// TIA Portal project "NeuroPLC_S7_1200_DB" (V21)

(* hardware
DEVICE "PLC_1"  S7-1200 Station
   slot 0: "Rack_0"  S7-1200 Rack  Rack  V1.0
   slot 1: "PLC_1"  CPU 1211C AC/DC/Rly  6ES7 211-1BE40-0XB0  V4.7
*)

// ===== PLC "PLC_1"  CPU 1211C AC/DC/Rly =====

DATA_BLOCK "NeuroPLC_KAN_Weights"   // DB1
{ S7_Optimized_Access := 'FALSE' }
VERSION : 0.1
   VAR
      g0 : Array[0..14] of Real;   // LUT grid (15 pts)
      t1 : Array[0..6719] of Real;   // LUT table (16x28x15)
      w2 : Array[0..447] of Real;   // W(16x28)
      b3 : Array[0..15] of Real;   // bias(16)
      g4 : Array[0..14] of Real;   // LUT grid (15 pts)
      t5 : Array[0..959] of Real;   // LUT table (4x16x15)
      w6 : Array[0..63] of Real;   // W(4x16)
      b7 : Array[0..3] of Real;   // bias(4)
   END_VAR
BEGIN
   g0[0] := -3.0;
   g0[1] := -2.571429;
   g0[2] := -2.142857;
   g0[3] := -1.714286;
   g0[4] := -1.285714;
   g0[5] := -0.8571429;
   g0[6] := -0.4285714;
   g0[8] := 0.4285714;
   g0[9] := 0.8571429;
   g0[10] := 1.285714;
   g0[11] := 1.714286;
   g0[12] := 2.142857;
   g0[13] := 2.571429;
   g0[14] := 3.0;
   t1[0] := -0.1194829;
   t1[1] := -0.1267372;
   t1[2] := -0.1291282;
   t1[3] := -0.1263348;
   t1[4] := -0.1178586;
   t1[5] := -0.1031384;
   t1[6] := -0.0816128;
   t1[7] := -0.0527206;
   t1[8] := -0.0159457;
   t1[9] := 0.0269625;
   t1[10] := 0.0709812;
   t1[11] := 0.1108319;
   t1[12] := 0.141236;
   t1[13] := 0.156915;
   t1[14] := 0.1536715;
   t1[15] := -0.0048413;
   t1[16] := -0.0066063;
   t1[17] := -0.0042641;
   t1[18] := 0.0032827;
   t1[19] := 0.0154041;
   t1[20] := 0.0308592;
   t1[21] := 0.0484067;
   t1[22] := 0.0668051;
   t1[23] := 0.0848193;
   t1[24] := 0.1015272;
   t1[25] := 0.1164593;
   t1[26] := 0.1291814;
   t1[27] := 0.1392594;
   t1[28] := 0.1462591;
   t1[29] := 0.1498416;
   t1[30] := -0.08693;
   t1[31] := -0.0833493;
   t1[32] := -0.0687987;
   t1[33] := -0.0417966;
   t1[34] := -0.0053218;
   t1[35] := 0.0360709;
   t1[36] := 0.0778248;
   t1[37] := 0.1153831;
   t1[38] := 0.144237;
   t1[39] := 0.1622724;
   t1[40] := 0.1708359;
   t1[41] := 0.1715441;
   t1[42] := 0.166014;
   t1[43] := 0.1558621;
   t1[44] := 0.1426646;
   t1[45] := -0.0762567;
   t1[46] := -0.0843287;
   t1[47] := -0.0897336;
   t1[48] := -0.0919366;
   t1[49] := -0.0903113;
   t1[50] := -0.0841991;
   t1[51] := -0.0729412;
   t1[52] := -0.055879;
   t1[53] := -0.0323818;
   t1[54] := -0.0032285;
   t1[55] := 0.0287655;
   t1[56] := 0.0606256;
   t1[57] := 0.0893772;
   t1[58] := 0.1120458;
   t1[59] := 0.1260427;
   t1[60] := -0.1835549;
   t1[61] := -0.1948409;
   t1[62] := -0.1973169;
   t1[63] := -0.1890172;
   t1[64] := -0.1712564;
   t1[65] := -0.1465084;
   t1[66] := -0.1172482;
   t1[67] := -0.0859511;
   t1[68] := -0.055075;
   t1[69] := -0.0262112;
   t1[70] := 0.000301;
   t1[71] := 0.0242203;
   t1[72] := 0.0453052;
   t1[73] := 0.0633144;
   t1[74] := 0.077947;
   t1[75] := -0.0558672;
   t1[76] := -0.0577179;
   t1[77] := -0.0553535;
   t1[78] := -0.0488306;
   t1[79] := -0.0385897;
   t1[80] := -0.025207;
   t1[81] := -0.0092587;
   t1[82] := 0.008679;
   t1[83] := 0.02802;
   t1[84] := 0.0476948;
   t1[85] := 0.0659345;
   t1[86] := 0.0809157;
   t1[87] := 0.0908151;
   t1[88] := 0.0938092;
   t1[89] := 0.0884755;
   t1[90] := 0.1269326;
   t1[91] := 0.1441061;
   t1[92] := 0.1569568;
   t1[93] := 0.1633429;
   t1[94] := 0.1623842;
   t1[95] := 0.153646;
   t1[96] := 0.1366941;
   t1[97] := 0.1110945;
   t1[98] := 0.0764416;
   t1[99] := 0.0337616;
   t1[100] := -0.0138503;
   t1[101] := -0.0631375;
   t1[102] := -0.1108431;
   t1[103] := -0.1537104;
   t1[104] := -0.1886999;
   t1[105] := -0.0070284;
   t1[106] := -0.0404032;
   t1[107] := -0.064115;
   t1[108] := -0.07382;
   t1[109] := -0.0709769;
   t1[110] := -0.0590946;
   t1[111] := -0.0416847;
   t1[112] := -0.0222583;
   t1[113] := -0.0042989;
   t1[114] := 0.0101144;
   t1[115] := 0.0209318;
   t1[116] := 0.0282619;
   t1[117] := 0.0322132;
   t1[118] := 0.0328943;
   t1[119] := 0.0304549;
   t1[120] := -0.1028974;
   t1[121] := -0.1077723;
   t1[122] := -0.1036677;
   t1[123] := -0.0897878;
   t1[124] := -0.0682854;
   t1[125] := -0.0423547;
   t1[126] := -0.0151914;
   t1[127] := 0.0100092;
   t1[128] := 0.030083;
   t1[129] := 0.0434435;
   t1[130] := 0.0507842;
   t1[131] := 0.0529767;
   t1[132] := 0.0508923;
   t1[133] := 0.0454027;
   t1[134] := 0.0373401;
   t1[135] := 0.0462424;
   t1[136] := 0.0249232;
   t1[137] := 0.0137322;
   t1[138] := 0.0163544;
   t1[139] := 0.0313536;
   t1[140] := 0.0554837;
   t1[141] := 0.0854967;
   t1[142] := 0.1181446;
   t1[143] := 0.1501878;
   t1[144] := 0.1788067;
   t1[145] := 0.2017891;
   t1[146] := 0.2169701;
   t1[147] := 0.2221848;
   t1[148] := 0.2152684;
   t1[149] := 0.1947507;
   t1[150] := 0.2054697;
   t1[151] := 0.1801361;
   t1[152] := 0.1482858;
   t1[153] := 0.1121279;
   t1[154] := 0.0745698;
   t1[155] := 0.0387658;
   t1[156] := 0.0078706;
   t1[157] := -0.0149613;
   t1[158] := -0.0266352;
   t1[159] := -0.0270458;
   t1[160] := -0.0204089;
   t1[161] := -0.0112777;
   t1[162] := -0.0042051;
   t1[163] := -0.0037442;
   t1[164] := -0.0135843;
   t1[165] := 0.069604;
   t1[166] := 0.0267136;
   t1[167] := -0.0201817;
   t1[168] := -0.0687582;
   t1[169] := -0.1154626;
   t1[170] := -0.156307;
   t1[171] := -0.1873028;
   t1[172] := -0.2044615;
   t1[173] := -0.2038705;
   t1[174] := -0.1854049;
   t1[175] := -0.1544143;
   t1[176] := -0.1166757;
   t1[177] := -0.0779662;
   t1[178] := -0.0440626;
   t1[179] := -0.0199858;
   t1[180] := 0.2695681;
   t1[181] := 0.2165021;
   t1[182] := 0.1619561;
   t1[183] := 0.1091502;
   t1[184] := 0.0593546;
   t1[185] := 0.0131512;
   t1[186] := -0.0288789;
   t1[187] := -0.0661548;
   t1[188] := -0.0981051;
   t1[189] := -0.1246367;
   t1[190] := -0.146348;
   t1[191] := -0.1638913;
   t1[192] := -0.177919;
   t1[193] := -0.1890834;
   t1[194] := -0.1978753;
   t1[195] := 0.1005199;
   t1[196] := 0.1037989;
   t1[197] := 0.1110083;
   t1[198] := 0.1225618;
   t1[199] := 0.1376169;
   t1[200] := 0.1548869;
   t1[201] := 0.1730847;
   t1[202] := 0.1909233;
   t1[203] := 0.2071245;
   t1[204] := 0.2208622;
   t1[205] := 0.231963;
   t1[206] := 0.2403047;
   t1[207] := 0.2457651;
   t1[208] := 0.2482219;
   t1[209] := 0.247544;
   t1[210] := 0.0554956;
   t1[211] := 0.0007121;
   t1[212] := -0.0460094;
   t1[213] := -0.078633;
   t1[214] := -0.0985512;
   t1[215] := -0.1097806;
   t1[216] := -0.1163414;
   t1[217] := -0.1222533;
   t1[218] := -0.1314804;
   t1[219] := -0.1451906;
   t1[220] := -0.1605101;
   t1[221] := -0.1742501;
   t1[222] := -0.1832213;
   t1[223] := -0.1842349;
   t1[224] := -0.1747214;
   t1[225] := -0.0316489;
   t1[226] := -0.0383947;
   t1[227] := -0.0447371;
   t1[228] := -0.0514102;
   t1[229] := -0.0574886;
   t1[230] := -0.0614606;
   t1[231] := -0.0618138;
   t1[232] := -0.0570359;
   t1[233] := -0.045655;
   t1[234] := -0.0282333;
   t1[235] := -0.0082723;
   t1[236] := 0.010497;
   t1[237] := 0.0243434;
   t1[238] := 0.0295361;
   t1[239] := 0.0231194;
   t1[240] := -0.0541978;
   t1[241] := -0.0262211;
   t1[242] := 0.0058194;
   t1[243] := 0.0394106;
   t1[244] := 0.0729769;
   t1[245] := 0.1052741;
   t1[246] := 0.1350584;
   t1[247] := 0.161086;
   t1[248] := 0.1821203;
   t1[249] := 0.1972881;
   t1[250] := 0.2062417;
   t1[251] := 0.208674;
   t1[252] := 0.2042782;
   t1[253] := 0.1927473;
   t1[254] := 0.1740892;
   t1[255] := 0.0165106;
   t1[256] := 0.0038278;
   t1[257] := -0.0110902;
   t1[258] := -0.0267964;
   t1[259] := -0.0414656;
   t1[260] := -0.0531389;
   t1[261] := -0.059857;
   t1[262] := -0.0596609;
   t1[263] := -0.050625;
   t1[264] := -0.0325026;
   t1[265] := -0.0074732;
   t1[266] := 0.0220942;
   t1[267] := 0.0538307;
   t1[268] := 0.0853673;
   t1[269] := 0.1144174;
   t1[270] := 0.2570028;
   t1[271] := 0.2134718;
   t1[272] := 0.1650651;
   t1[273] := 0.1143154;
   t1[274] := 0.0630908;
   t1[275] := 0.0130241;
   t1[276] := -0.0342518;
   t1[277] := -0.0771044;
   t1[278] := -0.1139093;
   t1[279] := -0.1434596;
   t1[280] := -0.1651517;
   t1[281] := -0.1784292;
   t1[282] := -0.1827355;
   t1[283] := -0.1775142;
   t1[284] := -0.1625242;
   t1[285] := 0.1695031;
   t1[286] := 0.1470198;
   t1[287] := 0.1199536;
   t1[288] := 0.0881358;
   t1[289] := 0.0530191;
   t1[290] := 0.0166294;
   t1[291] := -0.0190068;
   t1[292] := -0.051863;
   t1[293] := -0.0799368;
   t1[294] := -0.1024416;
   t1[295] := -0.1203473;
   t1[296] := -0.1347608;
   t1[297] := -0.1467892;
   t1[298] := -0.1575395;
   t1[299] := -0.1678591;
   t1[300] := -0.189392;
   t1[301] := -0.1452939;
   t1[302] := -0.1035419;
   t1[303] := -0.0676707;
   t1[304] := -0.0367318;
   t1[305] := -0.0081925;
   t1[306] := 0.0204816;
   t1[307] := 0.0518252;
   t1[308] := 0.0883329;
   t1[309] := 0.1305132;
   t1[310] := 0.1760034;
   t1[311] := 0.2222168;
   t1[312] := 0.2665667;
   t1[313] := 0.3064664;
   t1[314] := 0.3394241;
   t1[315] := -0.0330082;
   t1[316] := -0.0595727;
   t1[317] := -0.0757542;
   t1[318] := -0.0766687;
   t1[319] := -0.0640394;
   t1[320] := -0.0419239;
   t1[321] := -0.0143825;
   t1[322] := 0.0145245;
   t1[323] := 0.0407725;
   t1[324] := 0.0621279;
   t1[325] := 0.0789453;
   t1[326] := 0.0917811;
   t1[327] := 0.101192;
   t1[328] := 0.1077346;
   t1[329] := 0.1118888;
   t1[330] := -0.0263191;
   t1[331] := 0.0124622;
   t1[332] := 0.0404122;
   t1[333] := 0.0524193;
   t1[334] := 0.0510294;
   t1[335] := 0.0414941;
   t1[336] := 0.0290681;
   t1[337] := 0.019006;
   t1[338] := 0.0165029;
   t1[339] := 0.0237657;
   t1[340] := 0.0386827;
   t1[341] := 0.0588053;
   t1[342] := 0.0816847;
   t1[343] := 0.1048722;
   t1[344] := 0.1260335;
   t1[345] := 0.0412466;
   t1[346] := 0.0436516;
   t1[347] := 0.0403802;
   t1[348] := 0.031226;
   t1[349] := 0.018012;
   t1[350] := 0.0032783;
   t1[351] := -0.010434;
   t1[352] := -0.0205838;
   t1[353] := -0.0246632;
   t1[354] := -0.0218213;
   t1[355] := -0.0136019;
   t1[356] := -0.0017359;
   t1[357] := 0.0120461;
   t1[358] := 0.0260132;
   t1[359] := 0.0385597;
   t1[360] := 0.1668451;
   t1[361] := 0.1318458;
   t1[362] := 0.0940298;
   t1[363] := 0.0566781;
   t1[364] := 0.0218116;
   t1[365] := -0.0089939;
   t1[366] := -0.0341632;
   t1[367] := -0.052121;
   t1[368] := -0.0613163;
   t1[369] := -0.0614061;
   t1[370] := -0.0537936;
   t1[371] := -0.0400181;
   t1[372] := -0.0216192;
   t1[373] := -0.0001363;
   t1[374] := 0.0228733;
   t1[375] := -0.2291011;
   t1[376] := -0.2048234;
   t1[377] := -0.1736495;
   t1[378] := -0.1362531;
   t1[379] := -0.0941705;
   t1[380] := -0.049243;
   t1[381] := -0.0033123;
   t1[382] := 0.0417801;
   t1[383] := 0.0841977;
   t1[384] := 0.122365;
   t1[385] := 0.1550836;
   t1[386] := 0.1811845;
   t1[387] := 0.1994988;
   t1[388] := 0.2088575;
   t1[389] := 0.2084018;
   t1[390] := 0.0971736;
   t1[391] := 0.0705846;
   t1[392] := 0.0477992;
   t1[393] := 0.0314683;
   t1[394] := 0.0213695;
   t1[395] := 0.0162659;
   t1[396] := 0.014919;
   t1[397] := 0.0160906;
   t1[398] := 0.0185539;
   t1[399] := 0.0216598;
   t1[400] := 0.0255942;
   t1[401] := 0.0306081;
   t1[402] := 0.0369525;
   t1[403] := 0.0448785;
   t1[404] := 0.0544655;
   t1[405] := 0.1530943;
   t1[406] := 0.1480777;
   t1[407] := 0.1306549;
   t1[408] := 0.0980344;
   t1[409] := 0.0543566;
   t1[410] := 0.0062115;
   t1[411] := -0.0398084;
   t1[412] := -0.0771103;
   t1[413] := -0.0991863;
   t1[414] := -0.1037752;
   t1[415] := -0.0947527;
   t1[416] := -0.0764738;
   t1[417] := -0.0532932;
   t1[418] := -0.0295659;
   t1[419] := -0.0091988;
   t1[420] := -0.1092411;
   t1[421] := -0.1059756;
   t1[422] := -0.0969084;
   t1[423] := -0.0807166;
   t1[424] := -0.0580724;
   t1[425] := -0.0303529;
   t1[426] := 0.0010639;
   t1[427] := 0.0348003;
   t1[428] := 0.0694891;
   t1[429] := 0.1043026;
   t1[430] := 0.1391932;
   t1[431] := 0.1741739;
   t1[432] := 0.2092578;
   t1[433] := 0.2444581;
   t1[434] := 0.2795447;
   t1[435] := -0.1311382;
   t1[436] := -0.1227978;
   t1[437] := -0.1088914;
   t1[438] := -0.0897558;
   t1[439] := -0.0661454;
   t1[440] := -0.0389617;
   t1[441] := -0.0091066;
   t1[442] := 0.0225182;
   t1[443] := 0.0550137;
   t1[444] := 0.0876197;
   t1[445] := 0.1197764;
   t1[446] := 0.15094;
   t1[447] := 0.1805664;
   t1[448] := 0.2081117;
   t1[449] := 0.232934;
   t1[450] := -0.2517078;
   t1[451] := -0.2631014;
   t1[452] := -0.2655013;
   t1[453] := -0.2574791;
   t1[454] := -0.2394219;
   t1[455] := -0.2123581;
   t1[456] := -0.1773168;
   t1[457] := -0.1353271;
   t1[458] := -0.0874226;
   t1[459] := -0.0348577;
   t1[460] := 0.0207941;
   t1[461] := 0.0779343;
   t1[462] := 0.1349643;
   t1[463] := 0.1902857;
   t1[464] := 0.2421744;
   t1[465] := 0.0492069;
   t1[466] := 0.0399185;
   t1[467] := 0.0213245;
   t1[468] := -0.0083821;
   t1[469] := -0.0462682;
   t1[470] := -0.0877257;
   t1[471] := -0.1281447;
   t1[472] := -0.1629154;
   t1[473] := -0.187479;
   t1[474] := -0.1998351;
   t1[475] := -0.2016807;
   t1[476] := -0.1950018;
   t1[477] := -0.181784;
   t1[478] := -0.164013;
   t1[479] := -0.1435986;
   t1[480] := 0.2468299;
   t1[481] := 0.2682943;
   t1[482] := 0.2761828;
   t1[483] := 0.2661327;
   t1[484] := 0.2398228;
   t1[485] := 0.2010666;
   t1[486] := 0.1536797;
   t1[487] := 0.1014783;
   t1[488] := 0.0482628;
   t1[489] := -0.0029272;
   t1[490] := -0.0501526;
   t1[491] := -0.0915597;
   t1[492] := -0.1252953;
   t1[493] := -0.149506;
   t1[494] := -0.1626064;
   t1[495] := -0.0399078;
   t1[496] := -0.0051029;
   t1[497] := 0.0288762;
   t1[498] := 0.0581392;
   t1[499] := 0.0810207;
   t1[500] := 0.0966417;
   t1[501] := 0.1041238;
   t1[502] := 0.1025889;
   t1[503] := 0.0911945;
   t1[504] := 0.0708923;
   t1[505] := 0.0452268;
   t1[506] := 0.0179449;
   t1[507] := -0.0072066;
   t1[508] := -0.0264807;
   t1[509] := -0.0367556;
   t1[510] := -0.227583;
   t1[511] := -0.2168898;
   t1[512] := -0.2061395;
   t1[513] := -0.197567;
   t1[514] := -0.1891667;
   t1[515] := -0.1774349;
   t1[516] := -0.1588662;
   t1[517] := -0.129955;
   t1[518] := -0.0872722;
   t1[519] := -0.0312042;
   t1[520] := 0.0323485;
   t1[521] := 0.0970544;
   t1[522] := 0.1565824;
   t1[523] := 0.2046015;
   t1[524] := 0.235604;
   t1[525] := 0.15399;
   t1[526] := 0.1505588;
   t1[527] := 0.1378421;
   t1[528] := 0.1147972;
   t1[529] := 0.084201;
   t1[530] := 0.0501803;
   t1[531] := 0.0168631;
   t1[532] := -0.0116225;
   t1[533] := -0.0311856;
   t1[534] := -0.0396094;
   t1[535] := -0.0373845;
   t1[536] := -0.0252131;
   t1[537] := -0.0037974;
   t1[538] := 0.0261603;
   t1[539] := 0.063599;
   t1[540] := -0.1692545;
   t1[541] := -0.1745036;
   t1[542] := -0.1656465;
   t1[543] := -0.1392908;
   t1[544] := -0.099259;
   t1[545] := -0.0519229;
   t1[546] := -0.0036572;
   t1[547] := 0.0391633;
   t1[548] := 0.0702438;
   t1[549] := 0.087294;
   t1[550] := 0.0938102;
   t1[551] := 0.0937407;
   t1[552] := 0.091034;
   t1[553] := 0.0896381;
   t1[554] := 0.0929436;
   t1[555] := -0.1842585;
   t1[556] := -0.1818165;
   t1[557] := -0.1727193;
   t1[558] := -0.154162;
   t1[559] := -0.126589;
   t1[560] := -0.0915928;
   t1[561] := -0.050767;
   t1[562] := -0.0057056;
   t1[563] := 0.0420004;
   t1[564] := 0.0908896;
   t1[565] := 0.1396887;
   t1[566] := 0.1871389;
   t1[567] := 0.2319812;
   t1[568] := 0.272957;
   t1[569] := 0.3087583;
   t1[570] := -0.3433722;
   t1[571] := -0.3115804;
   t1[572] := -0.2701057;
   t1[573] := -0.2195741;
   t1[574] := -0.1626008;
   t1[575] := -0.1025036;
   t1[576] := -0.0426015;
   t1[577] := 0.0137868;
   t1[578] := 0.0633724;
   t1[579] := 0.1043585;
   t1[580] := 0.1371047;
   t1[581] := 0.1621392;
   t1[582] := 0.17999;
   t1[583] := 0.1911852;
   t1[584] := 0.1962473;
   t1[585] := 0.0363517;
   t1[586] := 0.0190614;
   t1[587] := 0.0082236;
   t1[588] := 0.0071252;
   t1[589] := 0.0142321;
   t1[590] := 0.0263068;
   t1[591] := 0.0401099;
   t1[592] := 0.0524021;
   t1[593] := 0.059982;
   t1[594] := 0.0615569;
   t1[595] := 0.0585923;
   t1[596] := 0.0527691;
   t1[597] := 0.0457681;
   t1[598] := 0.0392702;
   t1[599] := 0.0347328;
   t1[600] := -0.2135215;
   t1[601] := -0.1584936;
   t1[602] := -0.0996131;
   t1[603] := -0.0401407;
   t1[604] := 0.0172358;
   t1[605] := 0.0700308;
   t1[606] := 0.1157594;
   t1[607] := 0.1519362;
   t1[608] := 0.1761245;
   t1[609] := 0.1883052;
   t1[610] := 0.1919536;
   t1[611] := 0.190818;
   t1[612] := 0.1886465;
   t1[613] := 0.1891873;
   t1[614] := 0.1954547;
   t1[615] := -0.2638247;
   t1[616] := -0.2262976;
   t1[617] := -0.181273;
   t1[618] := -0.1300747;
   t1[619] := -0.0758695;
   t1[620] := -0.0224759;
   t1[621] := 0.0262873;
   t1[622] := 0.066601;
   t1[623] := 0.0947028;
   t1[624] := 0.1096649;
   t1[625] := 0.114656;
   t1[626] := 0.1131646;
   t1[627] := 0.1086792;
   t1[628] := 0.1046883;
   t1[629] := 0.1041317;
   t1[630] := -0.0215827;
   t1[631] := -0.0225016;
   t1[632] := -0.0222959;
   t1[633] := -0.018404;
   t1[634] := -0.0125777;
   t1[635] := -0.0080928;
   t1[636] := -0.0082266;
   t1[637] := -0.0162568;
   t1[638] := -0.0353979;
   t1[639] := -0.0657176;
   t1[640] := -0.1027351;
   t1[641] := -0.1416151;
   t1[642] := -0.1775218;
   t1[643] := -0.2056196;
   t1[644] := -0.2217522;
   t1[645] := 0.0948695;
   t1[646] := 0.1189938;
   t1[647] := 0.1318502;
   t1[648] := 0.1305514;
   t1[649] := 0.1161173;
   t1[650] := 0.0909486;
   t1[651] := 0.0574476;
   t1[652] := 0.0180163;
   t1[653] := -0.0249446;
   t1[654] := -0.0691197;
   t1[655] := -0.1123164;
   t1[656] := -0.1523517;
   t1[657] := -0.1870427;
   t1[658] := -0.2142063;
   t1[659] := -0.2319627;
   t1[660] := 0.2239106;
   t1[661] := 0.2024928;
   t1[662] := 0.1690608;
   t1[663] := 0.1246878;
   t1[664] := 0.0722037;
   t1[665] := 0.0150594;
   t1[666] := -0.0432937;
   t1[667] := -0.0994042;
   t1[668] := -0.1498503;
   t1[669] := -0.1927032;
   t1[670] := -0.228191;
   t1[671] := -0.2567104;
   t1[672] := -0.278658;
   t1[673] := -0.2944305;
   t1[674] := -0.3043407;
   t1[675] := -0.210152;
   t1[676] := -0.1704469;
   t1[677] := -0.1309727;
   t1[678] := -0.0954248;
   t1[679] := -0.0645113;
   t1[680] := -0.0378848;
   t1[681] := -0.0151968;
   t1[682] := 0.0039014;
   t1[683] := 0.0197446;
   t1[684] := 0.0319798;
   t1[685] := 0.0392597;
   t1[686] := 0.0401597;
   t1[687] := 0.0332549;
   t1[688] := 0.0171205;
   t1[689] := -0.0090543;
   t1[690] := -0.2450845;
   t1[691] := -0.2073944;
   t1[692] := -0.1587359;
   t1[693] := -0.0981581;
   t1[694] := -0.0301329;
   t1[695] := 0.0389517;
   t1[696] := 0.1027057;
   t1[697] := 0.1547389;
   t1[698] := 0.1887307;
   t1[699] := 0.201844;
   t1[700] := 0.1962753;
   t1[701] := 0.1746144;
   t1[702] := 0.139451;
   t1[703] := 0.0933749;
   t1[704] := 0.0393236;
   t1[705] := -0.4248369;
   t1[706] := -0.3962753;
   t1[707] := -0.3550233;
   t1[708] := -0.3007319;
   t1[709] := -0.235328;
   t1[710] := -0.1615429;
   t1[711] := -0.0821088;
   t1[712] := 0.0002421;
   t1[713] := 0.0827594;
   t1[714] := 0.1617863;
   t1[715] := 0.2323554;
   t1[716] := 0.2893972;
   t1[717] := 0.327842;
   t1[718] := 0.3426206;
   t1[719] := 0.3299596;
   t1[720] := 0.3017888;
   t1[721] := 0.2690612;
   t1[722] := 0.2316348;
   t1[723] := 0.1906948;
   t1[724] := 0.1469425;
   t1[725] := 0.1009079;
   t1[726] := 0.0531211;
   t1[727] := 0.0041119;
   t1[728] := -0.0455605;
   t1[729] := -0.0938802;
   t1[730] := -0.136726;
   t1[731] := -0.1698123;
   t1[732] := -0.1888533;
   t1[733] := -0.1895635;
   t1[734] := -0.1688053;
   t1[735] := 0.2525824;
   t1[736] := 0.18621;
   t1[737] := 0.1176589;
   t1[738] := 0.051741;
   t1[739] := -0.0101694;
   t1[740] := -0.0679128;
   t1[741] := -0.121331;
   t1[742] := -0.1702659;
   t1[743] := -0.2145509;
   t1[744] := -0.2535933;
   t1[745] := -0.2861848;
   t1[746] := -0.3110689;
   t1[747] := -0.3269894;
   t1[748] := -0.3326899;
   t1[749] := -0.3272332;
   t1[750] := 0.1863346;
   t1[751] := 0.1608573;
   t1[752] := 0.1253638;
   t1[753] := 0.0792565;
   t1[754] := 0.0245148;
   t1[755] := -0.0359716;
   t1[756] := -0.0993121;
   t1[757] := -0.162616;
   t1[758] := -0.2229935;
   t1[759] := -0.2776099;
   t1[760] := -0.3237095;
   t1[761] := -0.3585427;
   t1[762] := -0.37936;
   t1[763] := -0.383412;
   t1[764] := -0.3686952;
   t1[765] := 0.0815692;
   t1[766] := 0.048889;
   t1[767] := 0.0186305;
   t1[768] := -0.0063527;
   t1[769] := -0.0252718;
   t1[770] := -0.0380674;
   t1[771] := -0.0446811;
   t1[772] := -0.0450545;
   t1[773] := -0.039138;
   t1[774] := -0.027325;
   t1[775] := -0.0106499;
   t1[776] := 0.0098032;
   t1[777] := 0.0329501;
   t1[778] := 0.0577068;
   t1[779] := 0.0828865;
   t1[780] := 0.0296985;
   t1[781] := 0.0293068;
   t1[782] := 0.0253197;
   t1[783] := 0.0168562;
   t1[784] := 0.0036509;
   t1[785] := -0.0143439;
   t1[786] := -0.0371757;
   t1[787] := -0.0648922;
   t1[788] := -0.0975138;
   t1[789] := -0.1337178;
   t1[790] := -0.1702395;
   t1[791] := -0.2036626;
   t1[792] := -0.230571;
   t1[793] := -0.2475483;
   t1[794] := -0.2517596;
   t1[795] := 0.2789594;
   t1[796] := 0.2455961;
   t1[797] := 0.1948428;
   t1[798] := 0.1237554;
   t1[799] := 0.0379211;
   t1[800] := -0.0540573;
   t1[801] := -0.1435741;
   t1[802] := -0.2220234;
   t1[803] := -0.2809054;
   t1[804] := -0.3170266;
   t1[805] := -0.3348626;
   t1[806] := -0.3394876;
   t1[807] := -0.3359756;
   t1[808] := -0.3294011;
   t1[809] := -0.3241007;
   t1[810] := -0.0089786;
   t1[811] := -0.0362744;
   t1[812] := -0.0592059;
   t1[813] := -0.0759042;
   t1[814] := -0.0867897;
   t1[815] := -0.0930913;
   t1[816] := -0.0960391;
   t1[817] := -0.0968631;
   t1[818] := -0.0967854;
   t1[819] := -0.096635;
   t1[820] := -0.0966729;
   t1[821] := -0.0971155;
   t1[822] := -0.0981794;
   t1[823] := -0.1000812;
   t1[824] := -0.1029065;
   t1[825] := 0.1839082;
   t1[826] := 0.1417683;
   t1[827] := 0.1001777;
   t1[828] := 0.0606095;
   t1[829] := 0.0235777;
   t1[830] := -0.0107424;
   t1[831] := -0.0421758;
   t1[832] := -0.0705477;
   t1[833] := -0.0956898;
   t1[834] := -0.1177712;
   t1[835] := -0.1374487;
   t1[836] := -0.1554168;
   t1[837] := -0.1723702;
   t1[838] := -0.1890035;
   t1[839] := -0.2057118;
   t1[840] := 0.129127;
   t1[841] := 0.1110444;
   t1[842] := 0.0881457;
   t1[843] := 0.0602059;
   t1[844] := 0.0294074;
   t1[845] := -0.0012173;
   t1[846] := -0.0286343;
   t1[847] := -0.0498099;
   t1[848] := -0.0617627;
   t1[849] := -0.0641271;
   t1[850] := -0.0603176;
   t1[851] := -0.0540441;
   t1[852] := -0.0490163;
   t1[853] := -0.0489441;
   t1[854] := -0.0567943;
   t1[855] := 0.1542486;
   t1[856] := 0.1565695;
   t1[857] := 0.1564502;
   t1[858] := 0.1521189;
   t1[859] := 0.1425956;
   t1[860] := 0.1271801;
   t1[861] := 0.1051726;
   t1[862] := 0.0758731;
   t1[863] := 0.0386272;
   t1[864] := -0.0049518;
   t1[865] := -0.0499728;
   t1[866] := -0.0912888;
   t1[867] := -0.1237528;
   t1[868] := -0.142218;
   t1[869] := -0.1424568;
   t1[870] := 0.2432433;
   t1[871] := 0.2138474;
   t1[872] := 0.1802735;
   t1[873] := 0.1440694;
   t1[874] := 0.1073077;
   t1[875] := 0.0722467;
   t1[876] := 0.0411446;
   t1[877] := 0.0162596;
   t1[878] := -0.0001807;
   t1[879] := -0.0074959;
   t1[880] := -0.007241;
   t1[881] := -0.0011456;
   t1[882] := 0.0090608;
   t1[883] := 0.0216487;
   t1[884] := 0.0349876;
   t1[885] := 0.0060134;
   t1[886] := 0.0130141;
   t1[887] := 0.0237696;
   t1[888] := 0.0376019;
   t1[889] := 0.0534102;
   t1[890] := 0.0699445;
   t1[891] := 0.0859543;
   t1[892] := 0.1001894;
   t1[893] := 0.111415;
   t1[894] := 0.1191774;
   t1[895] := 0.1241514;
   t1[896] := 0.1270998;
   t1[897] := 0.1287857;
   t1[898] := 0.129972;
   t1[899] := 0.1312302;
   t1[900] := 0.1256087;
   t1[901] := 0.1563205;
   t1[902] := 0.1742733;
   t1[903] := 0.1740982;
   t1[904] := 0.1577529;
   t1[905] := 0.1297838;
   t1[906] := 0.0947405;
   t1[907] := 0.0571723;
   t1[908] := 0.0216062;
   t1[909] := -0.0085694;
   t1[910] := -0.0316105;
   t1[911] := -0.0459015;
   t1[912] := -0.049827;
   t1[913] := -0.0417713;
   t1[914] := -0.0207005;
   t1[915] := 0.0231812;
   t1[916] := -8.79E-05;
   t1[917] := -0.0219202;
   t1[918] := -0.0408588;
   t1[919] := -0.0559851;
   t1[920] := -0.0665707;
   t1[921] := -0.0718874;
   t1[922] := -0.0712072;
   t1[923] := -0.0638269;
   t1[924] := -0.0503005;
   t1[925] := -0.0329986;
   t1[926] := -0.0144336;
   t1[927] := 0.0028822;
   t1[928] := 0.0164362;
   t1[929] := 0.0240322;
   t1[930] := -0.038803;
   t1[931] := -0.0486055;
   t1[932] := -0.0605563;
   t1[933] := -0.0756327;
   t1[934] := -0.0925168;
   t1[935] := -0.1090798;
   t1[936] := -0.1231917;
   t1[937] := -0.1327229;
   t1[938] := -0.1355845;
   t1[939] := -0.1317421;
   t1[940] := -0.1241293;
   t1[941] := -0.115912;
   t1[942] := -0.1102559;
   t1[943] := -0.1103266;
   t1[944] := -0.1186093;
   t1[945] := 0.0876806;
   t1[946] := 0.0631336;
   t1[947] := 0.0427845;
   t1[948] := 0.029061;
   t1[949] := 0.0215176;
   t1[950] := 0.0186934;
   t1[951] := 0.0191267;
   t1[952] := 0.0213555;
   t1[953] := 0.0239225;
   t1[954] := 0.0255944;
   t1[955] := 0.0254626;
   t1[956] := 0.0226434;
   t1[957] := 0.0162533;
   t1[958] := 0.0054088;
   t1[959] := -0.0104808;
   t1[960] := 0.156688;
   t1[961] := 0.1603846;
   t1[962] := 0.154632;
   t1[963] := 0.1365645;
   t1[964] := 0.1083499;
   t1[965] := 0.0739346;
   t1[966] := 0.037267;
   t1[967] := 0.0022954;
   t1[968] := -0.0270664;
   t1[969] := -0.0486369;
   t1[970] := -0.0627384;
   t1[971] := -0.0698887;
   t1[972] := -0.0706053;
   t1[973] := -0.0654061;
   t1[974] := -0.0549072;
   t1[975] := -0.031862;
   t1[976] := -0.0455655;
   t1[977] := -0.05899;
   t1[978] := -0.0719112;
   t1[979] := -0.0830013;
   t1[980] := -0.0905426;
   t1[981] := -0.0928171;
   t1[982] := -0.0881065;
   t1[983] := -0.0747269;
   t1[984] := -0.0527012;
   t1[985] := -0.024519;
   t1[986] := 0.0071373;
   t1[987] := 0.0395853;
   t1[988] := 0.0701428;
   t1[989] := 0.0964227;
   t1[990] := -0.0839461;
   t1[991] := -0.0576546;
   t1[992] := -0.0354264;
   t1[993] := -0.0196391;
   t1[994] := -0.0088567;
   t1[995] := -0.0002962;
   t1[996] := 0.0088271;
   t1[997] := 0.0212979;
   t1[998] := 0.0398612;
   t1[999] := 0.065273;
   t1[1000] := 0.0954149;
   t1[1001] := 0.1279444;
   t1[1002] := 0.1605185;
   t1[1003] := 0.1907948;
   t1[1004] := 0.2165315;
   t1[1005] := -0.0905587;
   t1[1006] := -0.0770747;
   t1[1007] := -0.0567213;
   t1[1008] := -0.0278872;
   t1[1009] := 0.0072464;
   t1[1010] := 0.0451578;
   t1[1011] := 0.0823241;
   t1[1012] := 0.1152222;
   t1[1013] := 0.1403646;
   t1[1014] := 0.1560475;
   t1[1015] := 0.163145;
   t1[1016] := 0.1627322;
   t1[1017] := 0.1558844;
   t1[1018] := 0.1436767;
   t1[1019] := 0.127186;
   t1[1020] := 0.0801389;
   t1[1021] := 0.0963834;
   t1[1022] := 0.108559;
   t1[1023] := 0.1157784;
   t1[1024] := 0.118301;
   t1[1025] := 0.1167915;
   t1[1026] := 0.1119149;
   t1[1027] := 0.1043363;
   t1[1028] := 0.0947118;
   t1[1029] := 0.0832515;
   t1[1030] := 0.0695204;
   t1[1031] := 0.053033;
   t1[1032] := 0.033304;
   t1[1033] := 0.0098482;
   t1[1034] := -0.0174747;
   t1[1035] := -0.1516485;
   t1[1036] := -0.1540985;
   t1[1037] := -0.1466674;
   t1[1038] := -0.1275958;
   t1[1039] := -0.0997078;
   t1[1040] := -0.0674472;
   t1[1041] := -0.0352591;
   t1[1042] := -0.0075892;
   t1[1043] := 0.0111756;
   t1[1044] := 0.0195666;
   t1[1045] := 0.0203332;
   t1[1046] := 0.016554;
   t1[1047] := 0.0113074;
   t1[1048] := 0.0076722;
   t1[1049] := 0.008225;
   t1[1050] := 0.0634489;
   t1[1051] := 0.0811783;
   t1[1052] := 0.0962268;
   t1[1053] := 0.10831;
   t1[1054] := 0.1167574;
   t1[1055] := 0.1207618;
   t1[1056] := 0.1195159;
   t1[1057] := 0.1122126;
   t1[1058] := 0.098064;
   t1[1059] := 0.0772594;
   t1[1060] := 0.0514001;
   t1[1061] := 0.0221976;
   t1[1062] := -0.0086368;
   t1[1063] := -0.0393915;
   t1[1064] := -0.0683924;
   t1[1065] := 0.1123488;
   t1[1066] := 0.1230779;
   t1[1067] := 0.1300773;
   t1[1068] := 0.1324327;
   t1[1069] := 0.1300538;
   t1[1070] := 0.1231414;
   t1[1071] := 0.1118965;
   t1[1072] := 0.0965201;
   t1[1073] := 0.0772214;
   t1[1074] := 0.0546004;
   t1[1075] := 0.0298231;
   t1[1076] := 0.0040996;
   t1[1077] := -0.0213601;
   t1[1078] := -0.0453459;
   t1[1079] := -0.0666947;
   t1[1080] := 0.086788;
   t1[1081] := 0.0857459;
   t1[1082] := 0.0790944;
   t1[1083] := 0.0659556;
   t1[1084] := 0.0473873;
   t1[1085] := 0.0251316;
   t1[1086] := 0.0009313;
   t1[1087] := -0.0234709;
   t1[1088] := -0.0463343;
   t1[1089] := -0.0660255;
   t1[1090] := -0.0810656;
   t1[1091] := -0.089988;
   t1[1092] := -0.0913262;
   t1[1093] := -0.0836134;
   t1[1094] := -0.065901;
   t1[1095] := -0.2284766;
   t1[1096] := -0.2127118;
   t1[1097] := -0.1930615;
   t1[1098] := -0.1704066;
   t1[1099] := -0.1452529;
   t1[1100] := -0.1179738;
   t1[1101] := -0.0889426;
   t1[1102] := -0.0585324;
   t1[1103] := -0.0271343;
   t1[1104] := 0.0039699;
   t1[1105] := 0.0322105;
   t1[1106] := 0.0549177;
   t1[1107] := 0.0694212;
   t1[1108] := 0.0730513;
   t1[1109] := 0.0638202;
   t1[1110] := 0.2277943;
   t1[1111] := 0.1997769;
   t1[1112] := 0.1625425;
   t1[1113] := 0.1168391;
   t1[1114] := 0.0645341;
   t1[1115] := 0.0078901;
   t1[1116] := -0.0508299;
   t1[1117] := -0.1093625;
   t1[1118] := -0.1654526;
   t1[1119] := -0.2172411;
   t1[1120] := -0.2634413;
   t1[1121] := -0.3028113;
   t1[1122] := -0.3341089;
   t1[1123] := -0.3560926;
   t1[1124] := -0.3677126;
   t1[1125] := -0.1244165;
   t1[1126] := -0.1280328;
   t1[1127] := -0.1142789;
   t1[1128] := -0.0792962;
   t1[1129] := -0.0295003;
   t1[1130] := 0.0250634;
   t1[1131] := 0.0743448;
   t1[1132] := 0.1082942;
   t1[1133] := 0.1170034;
   t1[1134] := 0.0976608;
   t1[1135] := 0.0577103;
   t1[1136] := 0.0053964;
   t1[1137] := -0.0510362;
   t1[1138] := -0.1033431;
   t1[1139] := -0.1442712;
   t1[1140] := -0.2164453;
   t1[1141] := -0.1878679;
   t1[1142] := -0.1530626;
   t1[1143] := -0.1125679;
   t1[1144] := -0.0669061;
   t1[1145] := -0.016594;
   t1[1146] := 0.0378515;
   t1[1147] := 0.0959136;
   t1[1148] := 0.1570459;
   t1[1149] := 0.2192149;
   t1[1150] := 0.2782384;
   t1[1151] := 0.3297664;
   t1[1152] := 0.3694488;
   t1[1153] := 0.3929358;
   t1[1154] := 0.3966911;
   t1[1155] := 0.0686965;
   t1[1156] := 0.0321014;
   t1[1157] := 0.0016967;
   t1[1158] := -0.0196487;
   t1[1159] := -0.0324024;
   t1[1160] := -0.0382107;
   t1[1161] := -0.0387212;
   t1[1162] := -0.0355818;
   t1[1163] := -0.0304228;
   t1[1164] := -0.0240163;
   t1[1165] := -0.0158928;
   t1[1166] := -0.0054865;
   t1[1167] := 0.0077688;
   t1[1168] := 0.0244392;
   t1[1169] := 0.0447654;
   t1[1170] := -0.0021481;
   t1[1171] := -0.014136;
   t1[1172] := -0.0223624;
   t1[1173] := -0.0235746;
   t1[1174] := -0.0180489;
   t1[1175] := -0.0073088;
   t1[1176] := 0.0071209;
   t1[1177] := 0.0237153;
   t1[1178] := 0.0409628;
   t1[1179] := 0.0580158;
   t1[1180] := 0.0749864;
   t1[1181] := 0.0920617;
   t1[1182] := 0.1094285;
   t1[1183] := 0.1272741;
   t1[1184] := 0.1455524;
   t1[1185] := -0.216501;
   t1[1186] := -0.1766151;
   t1[1187] := -0.1385338;
   t1[1188] := -0.1050993;
   t1[1189] := -0.0763241;
   t1[1190] := -0.0512208;
   t1[1191] := -0.0288007;
   t1[1192] := -0.0080752;
   t1[1193] := 0.0119309;
   t1[1194] := 0.0315228;
   t1[1195] := 0.0500373;
   t1[1196] := 0.0667356;
   t1[1197] := 0.080879;
   t1[1198] := 0.0917286;
   t1[1199] := 0.0986432;
   t1[1200] := -0.0746187;
   t1[1201] := -0.0717946;
   t1[1202] := -0.0710188;
   t1[1203] := -0.0715004;
   t1[1204] := -0.0724446;
   t1[1205] := -0.0730552;
   t1[1206] := -0.0725359;
   t1[1207] := -0.0700906;
   t1[1208] := -0.0649327;
   t1[1209] := -0.0567654;
   t1[1210] := -0.0459993;
   t1[1211] := -0.0331002;
   t1[1212] := -0.0185342;
   t1[1213] := -0.0027669;
   t1[1214] := 0.013648;
   t1[1215] := -0.066879;
   t1[1216] := -0.0283577;
   t1[1217] := 0.0090817;
   t1[1218] := 0.0422216;
   t1[1219] := 0.0697739;
   t1[1220] := 0.0911323;
   t1[1221] := 0.1056913;
   t1[1222] := 0.1128454;
   t1[1223] := 0.1120159;
   t1[1224] := 0.1039635;
   t1[1225] := 0.0913848;
   t1[1226] := 0.0771276;
   t1[1227] := 0.0640396;
   t1[1228] := 0.0549686;
   t1[1229] := 0.0522503;
   t1[1230] := 0.0454941;
   t1[1231] := 0.0613973;
   t1[1232] := 0.0682752;
   t1[1233] := 0.0663741;
   t1[1234] := 0.0586508;
   t1[1235] := 0.0490198;
   t1[1236] := 0.0413965;
   t1[1237] := 0.0396965;
   t1[1238] := 0.0477759;
   t1[1239] := 0.0665263;
   t1[1240] := 0.0925546;
   t1[1241] := 0.1221332;
   t1[1242] := 0.1515345;
   t1[1243] := 0.177031;
   t1[1244] := 0.1952834;
   t1[1245] := 0.2041488;
   t1[1246] := 0.1573575;
   t1[1247] := 0.1091614;
   t1[1248] := 0.0614568;
   t1[1249] := 0.0151901;
   t1[1250] := -0.0290273;
   t1[1251] := -0.0705849;
   t1[1252] := -0.1088718;
   t1[1253] := -0.1432736;
   t1[1254] := -0.1729859;
   t1[1255] := -0.1969304;
   t1[1256] := -0.2140072;
   t1[1257] := -0.2231164;
   t1[1258] := -0.2231583;
   t1[1259] := -0.2133855;
   t1[1260] := 0.2150663;
   t1[1261] := 0.1876653;
   t1[1262] := 0.1545088;
   t1[1263] := 0.1170022;
   t1[1264] := 0.0764197;
   t1[1265] := 0.0339888;
   t1[1266] := -0.0090627;
   t1[1267] := -0.0515071;
   t1[1268] := -0.0921205;
   t1[1269] := -0.1298595;
   t1[1270] := -0.1639418;
   t1[1271] := -0.1936056;
   t1[1272] := -0.218089;
   t1[1273] := -0.2366302;
   t1[1274] := -0.2485075;
   t1[1275] := 0.2414207;
   t1[1276] := 0.2225287;
   t1[1277] := 0.1931808;
   t1[1278] := 0.1527537;
   t1[1279] := 0.1035641;
   t1[1280] := 0.0489673;
   t1[1281] := -0.0076804;
   t1[1282] := -0.0630224;
   t1[1283] := -0.1137186;
   t1[1284] := -0.157253;
   t1[1285] := -0.1922998;
   t1[1286] := -0.2176265;
   t1[1287] := -0.2320003;
   t1[1288] := -0.2341887;
   t1[1289] := -0.2234196;
   t1[1290] := 0.2182729;
   t1[1291] := 0.1844119;
   t1[1292] := 0.1508107;
   t1[1293] := 0.1204758;
   t1[1294] := 0.0928297;
   t1[1295] := 0.0660287;
   t1[1296] := 0.0382277;
   t1[1297] := 0.0075815;
   t1[1298] := -0.0277114;
   t1[1299] := -0.067279;
   t1[1300] := -0.1076072;
   t1[1301] := -0.144937;
   t1[1302] := -0.1755089;
   t1[1303] := -0.195564;
   t1[1304] := -0.2019965;
   t1[1305] := 0.1156876;
   t1[1306] := 0.1007238;
   t1[1307] := 0.0799841;
   t1[1308] := 0.0533242;
   t1[1309] := 0.0228277;
   t1[1310] := -0.0086342;
   t1[1311] := -0.0381896;
   t1[1312] := -0.0629663;
   t1[1313] := -0.0801382;
   t1[1314] := -0.0891679;
   t1[1315] := -0.0928259;
   t1[1316] := -0.0941413;
   t1[1317] := -0.0961427;
   t1[1318] := -0.1018592;
   t1[1319] := -0.1136766;
   t1[1320] := 0.3676715;
   t1[1321] := 0.3711612;
   t1[1322] := 0.3522576;
   t1[1323] := 0.3079492;
   t1[1324] := 0.2428329;
   t1[1325] := 0.1641943;
   t1[1326] := 0.0793218;
   t1[1327] := -0.0044959;
   t1[1328] := -0.0800348;
   t1[1329] := -0.1432979;
   t1[1330] := -0.1949525;
   t1[1331] := -0.2360297;
   t1[1332] := -0.2675607;
   t1[1333] := -0.2905769;
   t1[1334] := -0.3059254;
   t1[1335] := 0.0961941;
   t1[1336] := 0.0903286;
   t1[1337] := 0.0890003;
   t1[1338] := 0.0939519;
   t1[1339] := 0.1024837;
   t1[1340] := 0.110326;
   t1[1341] := 0.1132075;
   t1[1342] := 0.1068568;
   t1[1343] := 0.087083;
   t1[1344] := 0.0537128;
   t1[1345] := 0.0123796;
   t1[1346] := -0.0308297;
   t1[1347] := -0.0698284;
   t1[1348] := -0.0985298;
   t1[1349] := -0.111827;
   t1[1350] := 0.2368123;
   t1[1351] := 0.2266839;
   t1[1352] := 0.2172155;
   t1[1353] := 0.2101848;
   t1[1354] := 0.2046047;
   t1[1355] := 0.1985113;
   t1[1356] := 0.1899394;
   t1[1357] := 0.176924;
   t1[1358] := 0.1575328;
   t1[1359] := 0.1314766;
   t1[1360] := 0.1008404;
   t1[1361] := 0.0678948;
   t1[1362] := 0.0349104;
   t1[1363] := 0.0041577;
   t1[1364] := -0.0222704;
   t1[1365] := 0.125632;
   t1[1366] := 0.1308341;
   t1[1367] := 0.1361611;
   t1[1368] := 0.1414702;
   t1[1369] := 0.1453366;
   t1[1370] := 0.1458822;
   t1[1371] := 0.1412284;
   t1[1372] := 0.1294966;
   t1[1373] := 0.1088527;
   t1[1374] := 0.07969;
   t1[1375] := 0.0456207;
   t1[1376] := 0.0105081;
   t1[1377] := -0.0217841;
   t1[1378] := -0.0473926;
   t1[1379] := -0.0630571;
   t1[1380] := 0.2329057;
   t1[1381] := 0.2182491;
   t1[1382] := 0.1876312;
   t1[1383] := 0.1387771;
   t1[1384] := 0.0748382;
   t1[1385] := 0.0008835;
   t1[1386] := -0.0780161;
   t1[1387] := -0.1567895;
   t1[1388] := -0.230386;
   t1[1389] := -0.2947705;
   t1[1390] := -0.3473763;
   t1[1391] := -0.3857511;
   t1[1392] := -0.4074424;
   t1[1393] := -0.4099982;
   t1[1394] := -0.3917492;
   t1[1395] := 0.1621147;
   t1[1396] := 0.1490201;
   t1[1397] := 0.1213881;
   t1[1398] := 0.0782657;
   t1[1399] := 0.025471;
   t1[1400] := -0.0287849;
   t1[1401] := -0.0762884;
   t1[1402] := -0.1088259;
   t1[1403] := -0.118307;
   t1[1404] := -0.1028219;
   t1[1405] := -0.0693925;
   t1[1406] := -0.0257379;
   t1[1407] := 0.0204228;
   t1[1408] := 0.0613705;
   t1[1409] := 0.0904432;
   t1[1410] := -0.1177829;
   t1[1411] := -0.1223881;
   t1[1412] := -0.1187199;
   t1[1413] := -0.1033856;
   t1[1414] := -0.0772939;
   t1[1415] := -0.0428736;
   t1[1416] := -0.0025552;
   t1[1417] := 0.0412309;
   t1[1418] := 0.0860618;
   t1[1419] := 0.129898;
   t1[1420] := 0.1712537;
   t1[1421] := 0.2086867;
   t1[1422] := 0.2407544;
   t1[1423] := 0.2660144;
   t1[1424] := 0.2831567;
   t1[1425] := -0.2121433;
   t1[1426] := -0.2094475;
   t1[1427] := -0.202064;
   t1[1428] := -0.1896108;
   t1[1429] := -0.1712027;
   t1[1430] := -0.1457771;
   t1[1431] := -0.1122708;
   t1[1432] := -0.0696208;
   t1[1433] := -0.0168151;
   t1[1434] := 0.044609;
   t1[1435] := 0.1094292;
   t1[1436] := 0.1721357;
   t1[1437] := 0.2272186;
   t1[1438] := 0.2691683;
   t1[1439] := 0.2932858;
   t1[1440] := -0.1129276;
   t1[1441] := -0.1059872;
   t1[1442] := -0.0913288;
   t1[1443] := -0.0668644;
   t1[1444] := -0.0344949;
   t1[1445] := 0.0024689;
   t1[1446] := 0.0407148;
   t1[1447] := 0.0769304;
   t1[1448] := 0.1078328;
   t1[1449] := 0.131597;
   t1[1450] := 0.1485059;
   t1[1451] := 0.1590068;
   t1[1452] := 0.163547;
   t1[1453] := 0.1625741;
   t1[1454] := 0.156581;
   t1[1455] := -0.0891135;
   t1[1456] := -0.0688476;
   t1[1457] := -0.0423377;
   t1[1458] := -0.0087247;
   t1[1459] := 0.0285992;
   t1[1460] := 0.0647393;
   t1[1461] := 0.0947991;
   t1[1462] := 0.1138824;
   t1[1463] := 0.1171789;
   t1[1464] := 0.1041952;
   t1[1465] := 0.080676;
   t1[1466] := 0.0528532;
   t1[1467] := 0.0269585;
   t1[1468] := 0.0092236;
   t1[1469] := 0.0048408;
   t1[1470] := 0.0594075;
   t1[1471] := 0.0981974;
   t1[1472] := 0.1312016;
   t1[1473] := 0.1565969;
   t1[1474] := 0.1739725;
   t1[1475] := 0.1834167;
   t1[1476] := 0.1850181;
   t1[1477] := 0.1788654;
   t1[1478] := 0.1650767;
   t1[1479] := 0.1452332;
   t1[1480] := 0.1230311;
   t1[1481] := 0.1023315;
   t1[1482] := 0.0869957;
   t1[1483] := 0.0808848;
   t1[1484] := 0.0869718;
   t1[1485] := -0.0385842;
   t1[1486] := -0.0422583;
   t1[1487] := -0.0356648;
   t1[1488] := -0.0150235;
   t1[1489] := 0.0169635;
   t1[1490] := 0.0553034;
   t1[1491] := 0.0950013;
   t1[1492] := 0.1310616;
   t1[1493] := 0.1585371;
   t1[1494] := 0.1748712;
   t1[1495] := 0.180963;
   t1[1496] := 0.1779814;
   t1[1497] := 0.1670951;
   t1[1498] := 0.149473;
   t1[1499] := 0.1263696;
   t1[1500] := 0.215929;
   t1[1501] := 0.1978684;
   t1[1502] := 0.1753161;
   t1[1503] := 0.1495115;
   t1[1504] := 0.1218254;
   t1[1505] := 0.0936746;
   t1[1506] := 0.0664763;
   t1[1507] := 0.0416473;
   t1[1508] := 0.0205874;
   t1[1509] := 0.0038223;
   t1[1510] := -0.0093854;
   t1[1511] := -0.0198714;
   t1[1512] := -0.0284716;
   t1[1513] := -0.0360217;
   t1[1514] := -0.043162;
   t1[1515] := -0.2822273;
   t1[1516] := -0.2620788;
   t1[1517] := -0.2337892;
   t1[1518] := -0.1974921;
   t1[1519] := -0.1545763;
   t1[1520] := -0.1068746;
   t1[1521] := -0.0562199;
   t1[1522] := -0.0044453;
   t1[1523] := 0.0466171;
   t1[1524] := 0.0951856;
   t1[1525] := 0.139551;
   t1[1526] := 0.1780101;
   t1[1527] := 0.2088594;
   t1[1528] := 0.2303957;
   t1[1529] := 0.2412203;
   t1[1530] := 0.1144546;
   t1[1531] := 0.0827512;
   t1[1532] := 0.0444258;
   t1[1533] := 0.0015962;
   t1[1534] := -0.0426917;
   t1[1535] := -0.0850639;
   t1[1536] := -0.1221464;
   t1[1537] := -0.1505648;
   t1[1538] := -0.166986;
   t1[1539] := -0.1701338;
   t1[1540] := -0.1617043;
   t1[1541] := -0.1436256;
   t1[1542] := -0.117826;
   t1[1543] := -0.0862338;
   t1[1544] := -0.0507871;
   t1[1545] := -0.2542355;
   t1[1546] := -0.2352409;
   t1[1547] := -0.2059316;
   t1[1548] := -0.1654823;
   t1[1549] := -0.1160405;
   t1[1550] := -0.060804;
   t1[1551] := -0.0029719;
   t1[1552] := 0.0542569;
   t1[1553] := 0.1076961;
   t1[1554] := 0.154797;
   t1[1555] := 0.1939323;
   t1[1556] := 0.2235466;
   t1[1557] := 0.2420845;
   t1[1558] := 0.2479907;
   t1[1559] := 0.2400402;
   t1[1560] := -0.0663666;
   t1[1561] := -0.0405909;
   t1[1562] := -0.0130403;
   t1[1563] := 0.0162417;
   t1[1564] := 0.0459971;
   t1[1565] := 0.0745388;
   t1[1566] := 0.1001791;
   t1[1567] := 0.1212304;
   t1[1568] := 0.1360299;
   t1[1569] := 0.1441571;
   t1[1570] := 0.1469874;
   t1[1571] := 0.1460363;
   t1[1572] := 0.1428191;
   t1[1573] := 0.1388514;
   t1[1574] := 0.1354096;
   t1[1575] := 0.1697915;
   t1[1576] := 0.1665091;
   t1[1577] := 0.1648042;
   t1[1578] := 0.16548;
   t1[1579] := 0.1676853;
   t1[1580] := 0.1699841;
   t1[1581] := 0.17094;
   t1[1582] := 0.1691164;
   t1[1583] := 0.163105;
   t1[1584] := 0.1529088;
   t1[1585] := 0.1405702;
   t1[1586] := 0.1282908;
   t1[1587] := 0.1182724;
   t1[1588] := 0.1127166;
   t1[1589] := 0.1133297;
   t1[1590] := -0.0068435;
   t1[1591] := 0.0184567;
   t1[1592] := 0.0357059;
   t1[1593] := 0.0410621;
   t1[1594] := 0.0363212;
   t1[1595] := 0.0252712;
   t1[1596] := 0.0117021;
   t1[1597] := -0.0005959;
   t1[1598] := -0.007872;
   t1[1599] := -0.0083354;
   t1[1600] := -0.0030287;
   t1[1601] := 0.0067844;
   t1[1602] := 0.0198403;
   t1[1603] := 0.0348752;
   t1[1604] := 0.0506105;
   t1[1605] := -0.1058745;
   t1[1606] := -0.0806083;
   t1[1607] := -0.0445283;
   t1[1608] := 0.005129;
   t1[1609] := 0.0642151;
   t1[1610] := 0.1261395;
   t1[1611] := 0.1843085;
   t1[1612] := 0.2321287;
   t1[1613] := 0.2630951;
   t1[1614] := 0.2751303;
   t1[1615] := 0.2725559;
   t1[1616] := 0.2601933;
   t1[1617] := 0.2428634;
   t1[1618] := 0.2253875;
   t1[1619] := 0.2119071;
   t1[1620] := -0.2206352;
   t1[1621] := -0.1945521;
   t1[1622] := -0.1603801;
   t1[1623] := -0.1170611;
   t1[1624] := -0.0675707;
   t1[1625] := -0.0163108;
   t1[1626] := 0.0323156;
   t1[1627] := 0.0739054;
   t1[1628] := 0.1041015;
   t1[1629] := 0.1208598;
   t1[1630] := 0.1254786;
   t1[1631] := 0.1195172;
   t1[1632] := 0.1045348;
   t1[1633] := 0.0820907;
   t1[1634] := 0.0538737;
   t1[1635] := -0.1020658;
   t1[1636] := -0.0799589;
   t1[1637] := -0.0544754;
   t1[1638] := -0.0253806;
   t1[1639] := 0.0065198;
   t1[1640] := 0.0400519;
   t1[1641] := 0.0740417;
   t1[1642] := 0.1073149;
   t1[1643] := 0.138701;
   t1[1644] := 0.1672044;
   t1[1645] := 0.1920826;
   t1[1646] := 0.2126128;
   t1[1647] := 0.2280724;
   t1[1648] := 0.2377387;
   t1[1649] := 0.2409902;
   t1[1650] := -0.3904826;
   t1[1651] := -0.3546944;
   t1[1652] := -0.3062641;
   t1[1653] := -0.2428138;
   t1[1654] := -0.1676919;
   t1[1655] := -0.0862703;
   t1[1656] := -0.0039232;
   t1[1657] := 0.0739752;
   t1[1658] := 0.1420963;
   t1[1659] := 0.1973947;
   t1[1660] := 0.2401244;
   t1[1661] := 0.2707972;
   t1[1662] := 0.2899245;
   t1[1663] := 0.2980182;
   t1[1664] := 0.2957028;
   t1[1665] := 0.0395081;
   t1[1666] := 0.0063693;
   t1[1667] := -0.0244155;
   t1[1668] := -0.052051;
   t1[1669] := -0.0748594;
   t1[1670] := -0.0908511;
   t1[1671] := -0.098036;
   t1[1672] := -0.0944242;
   t1[1673] := -0.0780796;
   t1[1674] := -0.0497685;
   t1[1675] := -0.0141629;
   t1[1676] := 0.0237604;
   t1[1677] := 0.0590247;
   t1[1678] := 0.0866533;
   t1[1679] := 0.1023997;
   t1[1680] := 0.1784618;
   t1[1681] := 0.200338;
   t1[1682] := 0.214846;
   t1[1683] := 0.2188044;
   t1[1684] := 0.2126888;
   t1[1685] := 0.1982669;
   t1[1686] := 0.177308;
   t1[1687] := 0.1515814;
   t1[1688] := 0.1228567;
   t1[1689] := 0.0929327;
   t1[1690] := 0.0636497;
   t1[1691] := 0.036851;
   t1[1692] := 0.0143803;
   t1[1693] := -0.0019189;
   t1[1694] := -0.0105719;
   t1[1695] := -0.0096433;
   t1[1696] := 0.0028053;
   t1[1697] := 0.0247683;
   t1[1698] := 0.0580469;
   t1[1699] := 0.0987041;
   t1[1700] := 0.1407751;
   t1[1701] := 0.1782929;
   t1[1702] := 0.2052903;
   t1[1703] := 0.2158899;
   t1[1704] := 0.2086912;
   t1[1705] := 0.1887638;
   t1[1706] := 0.1616829;
   t1[1707] := 0.1330232;
   t1[1708] := 0.1083599;
   t1[1709] := 0.0924743;
   t1[1710] := 0.0339864;
   t1[1711] := 0.030911;
   t1[1712] := 0.0288641;
   t1[1713] := 0.0280846;
   t1[1714] := 0.0278114;
   t1[1715] := 0.0269301;
   t1[1716] := 0.0243257;
   t1[1717] := 0.0188835;
   t1[1718] := 0.0095114;
   t1[1719] := -0.0037376;
   t1[1720] := -0.0191556;
   t1[1721] := -0.0349055;
   t1[1722] := -0.0491503;
   t1[1723] := -0.0600529;
   t1[1724] := -0.0660426;
   t1[1725] := -0.0108767;
   t1[1726] := 0.0006152;
   t1[1727] := 0.0122371;
   t1[1728] := 0.0229471;
   t1[1729] := 0.0327594;
   t1[1730] := 0.0420611;
   t1[1731] := 0.05124;
   t1[1732] := 0.0606839;
   t1[1733] := 0.0707736;
   t1[1734] := 0.0815549;
   t1[1735] := 0.0925886;
   t1[1736] := 0.1033979;
   t1[1737] := 0.1135058;
   t1[1738] := 0.1224356;
   t1[1739] := 0.129731;
   t1[1740] := 0.0594713;
   t1[1741] := 0.0477949;
   t1[1742] := 0.0380958;
   t1[1743] := 0.0330178;
   t1[1744] := 0.0323;
   t1[1745] := 0.0346555;
   t1[1746] := 0.0387961;
   t1[1747] := 0.0434335;
   t1[1748] := 0.0472924;
   t1[1749] := 0.0497408;
   t1[1750] := 0.0510765;
   t1[1751] := 0.0516699;
   t1[1752] := 0.0518913;
   t1[1753] := 0.0521111;
   t1[1754] := 0.0524928;
   t1[1755] := 0.0746827;
   t1[1756] := 0.0792039;
   t1[1757] := 0.0828199;
   t1[1758] := 0.0858207;
   t1[1759] := 0.0887841;
   t1[1760] := 0.0923895;
   t1[1761] := 0.0973166;
   t1[1762] := 0.104245;
   t1[1763] := 0.1138304;
   t1[1764] := 0.1255321;
   t1[1765] := 0.1370801;
   t1[1766] := 0.1460696;
   t1[1767] := 0.1500958;
   t1[1768] := 0.1467536;
   t1[1769] := 0.1341752;
   t1[1770] := 0.1423496;
   t1[1771] := 0.1520838;
   t1[1772] := 0.1638987;
   t1[1773] := 0.1785654;
   t1[1774] := 0.1945144;
   t1[1775] := 0.2093489;
   t1[1776] := 0.2206715;
   t1[1777] := 0.2260844;
   t1[1778] := 0.2232253;
   t1[1779] := 0.2114895;
   t1[1780] := 0.1928129;
   t1[1781] := 0.1693299;
   t1[1782] := 0.1431748;
   t1[1783] := 0.1164818;
   t1[1784] := 0.0912272;
   t1[1785] := 0.1119813;
   t1[1786] := 0.0956419;
   t1[1787] := 0.0816481;
   t1[1788] := 0.0724034;
   t1[1789] := 0.0667057;
   t1[1790] := 0.0620782;
   t1[1791] := 0.0560433;
   t1[1792] := 0.0461229;
   t1[1793] := 0.0298928;
   t1[1794] := 0.007623;
   t1[1795] := -0.0165236;
   t1[1796] := -0.03808;
   t1[1797] := -0.0525793;
   t1[1798] := -0.0555545;
   t1[1799] := -0.0435485;
   t1[1800] := 0.2142408;
   t1[1801] := 0.2057686;
   t1[1802] := 0.1967961;
   t1[1803] := 0.1890757;
   t1[1804] := 0.1818423;
   t1[1805] := 0.1734414;
   t1[1806] := 0.1622173;
   t1[1807] := 0.1465146;
   t1[1808] := 0.1247116;
   t1[1809] := 0.0968786;
   t1[1810] := 0.0655316;
   t1[1811] := 0.0333776;
   t1[1812] := 0.0031236;
   t1[1813] := -0.0225236;
   t1[1814] := -0.0412055;
   t1[1815] := 0.116414;
   t1[1816] := 0.1095619;
   t1[1817] := 0.1048087;
   t1[1818] := 0.1041354;
   t1[1819] := 0.1070599;
   t1[1820] := 0.1122296;
   t1[1821] := 0.1182909;
   t1[1822] := 0.1238903;
   t1[1823] := 0.1276824;
   t1[1824] := 0.1287377;
   t1[1825] := 0.1267277;
   t1[1826] := 0.1213706;
   t1[1827] := 0.1123848;
   t1[1828] := 0.0994885;
   t1[1829] := 0.0826378;
   t1[1830] := 0.0632413;
   t1[1831] := 0.0441744;
   t1[1832] := 0.0240819;
   t1[1833] := 0.0040768;
   t1[1834] := -0.0153211;
   t1[1835] := -0.0338016;
   t1[1836] := -0.0510549;
   t1[1837] := -0.0667712;
   t1[1838] := -0.0806448;
   t1[1839] := -0.0925765;
   t1[1840] := -0.102766;
   t1[1841] := -0.1114362;
   t1[1842] := -0.1188101;
   t1[1843] := -0.1251106;
   t1[1844] := -0.1304564;
   t1[1845] := 0.011329;
   t1[1846] := 0.0047532;
   t1[1847] := 0.0106199;
   t1[1848] := 0.03174;
   t1[1849] := 0.0640749;
   t1[1850] := 0.1011654;
   t1[1851] := 0.1365498;
   t1[1852] := 0.1637665;
   t1[1853] := 0.1764402;
   t1[1854] := 0.1725288;
   t1[1855] := 0.1562527;
   t1[1856] := 0.1323209;
   t1[1857] := 0.1054426;
   t1[1858] := 0.080327;
   t1[1859] := 0.0610837;
   t1[1860] := -0.0507518;
   t1[1861] := -0.0141973;
   t1[1862] := 0.0212375;
   t1[1863] := 0.0534648;
   t1[1864] := 0.0813056;
   t1[1865] := 0.1039018;
   t1[1866] := 0.120396;
   t1[1867] := 0.1299306;
   t1[1868] := 0.1316725;
   t1[1869] := 0.1260172;
   t1[1870] := 0.1151354;
   t1[1871] := 0.1013365;
   t1[1872] := 0.0869298;
   t1[1873] := 0.0742248;
   t1[1874] := 0.0652096;
   t1[1875] := -0.0238219;
   t1[1876] := -0.0227991;
   t1[1877] := -0.0212078;
   t1[1878] := -0.018609;
   t1[1879] := -0.0154283;
   t1[1880] := -0.0123966;
   t1[1881] := -0.0102453;
   t1[1882] := -0.0097058;
   t1[1883] := -0.0114932;
   t1[1884] := -0.0155161;
   t1[1885] := -0.0205174;
   t1[1886] := -0.025149;
   t1[1887] := -0.0280628;
   t1[1888] := -0.0279106;
   t1[1889] := -0.0236204;
   t1[1890] := 0.1261911;
   t1[1891] := 0.1180965;
   t1[1892] := 0.1095702;
   t1[1893] := 0.1010529;
   t1[1894] := 0.0933396;
   t1[1895] := 0.0873508;
   t1[1896] := 0.0840069;
   t1[1897] := 0.0842287;
   t1[1898] := 0.0889129;
   t1[1899] := 0.0977747;
   t1[1900] := 0.1088208;
   t1[1901] := 0.119925;
   t1[1902] := 0.1289607;
   t1[1903] := 0.1338014;
   t1[1904] := 0.1326779;
   t1[1905] := -0.2080787;
   t1[1906] := -0.1926835;
   t1[1907] := -0.1690558;
   t1[1908] := -0.1364757;
   t1[1909] := -0.0969082;
   t1[1910] := -0.0532668;
   t1[1911] := -0.0084665;
   t1[1912] := 0.034578;
   t1[1913] := 0.0729742;
   t1[1914] := 0.1049466;
   t1[1915] := 0.130334;
   t1[1916] := 0.149101;
   t1[1917] := 0.1612126;
   t1[1918] := 0.1666333;
   t1[1919] := 0.165435;
   t1[1920] := -0.0337367;
   t1[1921] := 0.0179158;
   t1[1922] := 0.0642252;
   t1[1923] := 0.100448;
   t1[1924] := 0.1261573;
   t1[1925] := 0.1424514;
   t1[1926] := 0.1504302;
   t1[1927] := 0.1511937;
   t1[1928] := 0.1458529;
   t1[1929] := 0.1360679;
   t1[1930] := 0.1242923;
   t1[1931] := 0.1130418;
   t1[1932] := 0.1048321;
   t1[1933] := 0.1021788;
   t1[1934] := 0.1069416;
   t1[1935] := 0.094077;
   t1[1936] := 0.0856499;
   t1[1937] := 0.0805157;
   t1[1938] := 0.0789634;
   t1[1939] := 0.0801158;
   t1[1940] := 0.0826838;
   t1[1941] := 0.0853779;
   t1[1942] := 0.0869084;
   t1[1943] := 0.0859976;
   t1[1944] := 0.0819534;
   t1[1945] := 0.0749302;
   t1[1946] := 0.0651486;
   t1[1947] := 0.0528292;
   t1[1948] := 0.0381926;
   t1[1949] := 0.0215873;
   t1[1950] := 0.0588603;
   t1[1951] := 0.0338434;
   t1[1952] := 0.0146228;
   t1[1953] := 0.0045955;
   t1[1954] := 0.0026677;
   t1[1955] := 0.0061591;
   t1[1956] := 0.0123873;
   t1[1957] := 0.0186702;
   t1[1958] := 0.0223601;
   t1[1959] := 0.022543;
   t1[1960] := 0.0208099;
   t1[1961] := 0.0189476;
   t1[1962] := 0.0187428;
   t1[1963] := 0.0219823;
   t1[1964] := 0.0300633;
   t1[1965] := 0.1109871;
   t1[1966] := 0.1151826;
   t1[1967] := 0.1166855;
   t1[1968] := 0.1157114;
   t1[1969] := 0.1126302;
   t1[1970] := 0.1078664;
   t1[1971] := 0.1018442;
   t1[1972] := 0.0949882;
   t1[1973] := 0.0877391;
   t1[1974] := 0.0813603;
   t1[1975] := 0.0783033;
   t1[1976] := 0.0811128;
   t1[1977] := 0.0923332;
   t1[1978] := 0.1145092;
   t1[1979] := 0.1493235;
   t1[1980] := 0.0914499;
   t1[1981] := 0.100605;
   t1[1982] := 0.1068323;
   t1[1983] := 0.1079146;
   t1[1984] := 0.1038054;
   t1[1985] := 0.0952249;
   t1[1986] := 0.0828944;
   t1[1987] := 0.067535;
   t1[1988] := 0.049871;
   t1[1989] := 0.0307813;
   t1[1990] := 0.0113679;
   t1[1991] := -0.0072493;
   t1[1992] := -0.0239508;
   t1[1993] := -0.0376169;
   t1[1994] := -0.0472918;
   t1[1995] := 0.0675064;
   t1[1996] := 0.0902898;
   t1[1997] := 0.1016986;
   t1[1998] := 0.1000157;
   t1[1999] := 0.0879783;
   t1[2000] := 0.0698969;
   t1[2001] := 0.0500841;
   t1[2002] := 0.0328523;
   t1[2003] := 0.022452;
   t1[2004] := 0.0200269;
   t1[2005] := 0.0222309;
   t1[2006] := 0.0253673;
   t1[2007] := 0.0257394;
   t1[2008] := 0.0196507;
   t1[2009] := 0.0041796;
   t1[2010] := 0.0393435;
   t1[2011] := 0.0357299;
   t1[2012] := 0.0373672;
   t1[2013] := 0.0463919;
   t1[2014] := 0.0610036;
   t1[2015] := 0.0780111;
   t1[2016] := 0.0942215;
   t1[2017] := 0.1064419;
   t1[2018] := 0.1115256;
   t1[2019] := 0.1086386;
   t1[2020] := 0.1002888;
   t1[2021] := 0.0892454;
   t1[2022] := 0.0782774;
   t1[2023] := 0.0701537;
   t1[2024] := 0.0671683;
   t1[2025] := 0.0297746;
   t1[2026] := 0.0581436;
   t1[2027] := 0.0834709;
   t1[2028] := 0.1041296;
   t1[2029] := 0.1202052;
   t1[2030] := 0.1323883;
   t1[2031] := 0.1413703;
   t1[2032] := 0.1478422;
   t1[2033] := 0.1524869;
   t1[2034] := 0.1555543;
   t1[2035] := 0.1566691;
   t1[2036] := 0.1554076;
   t1[2037] := 0.1513455;
   t1[2038] := 0.144059;
   t1[2039] := 0.1332652;
   t1[2040] := 0.3318817;
   t1[2041] := 0.3099373;
   t1[2042] := 0.2754277;
   t1[2043] := 0.2300242;
   t1[2044] := 0.177273;
   t1[2045] := 0.1213829;
   t1[2046] := 0.0665632;
   t1[2047] := 0.0170236;
   t1[2048] := -0.0230667;
   t1[2049] := -0.0515538;
   t1[2050] := -0.0691964;
   t1[2051] := -0.0769804;
   t1[2052] := -0.0758918;
   t1[2053] := -0.0669167;
   t1[2054] := -0.0512186;
   t1[2055] := 0.0525684;
   t1[2056] := 0.0687035;
   t1[2057] := 0.0862005;
   t1[2058] := 0.1057093;
   t1[2059] := 0.1256139;
   t1[2060] := 0.1434973;
   t1[2061] := 0.1569419;
   t1[2062] := 0.1635297;
   t1[2063] := 0.1608901;
   t1[2064] := 0.1490099;
   t1[2065] := 0.131283;
   t1[2066] := 0.1113693;
   t1[2067] := 0.0929287;
   t1[2068] := 0.079621;
   t1[2069] := 0.0744535;
   t1[2070] := 0.0967118;
   t1[2071] := 0.072273;
   t1[2072] := 0.0479304;
   t1[2073] := 0.024145;
   t1[2074] := 0.0027312;
   t1[2075] := -0.0140183;
   t1[2076] := -0.0238104;
   t1[2077] := -0.0243518;
   t1[2078] := -0.0134064;
   t1[2079] := 0.0084055;
   t1[2080] := 0.0363354;
   t1[2081] := 0.0653126;
   t1[2082] := 0.0902664;
   t1[2083] := 0.106126;
   t1[2084] := 0.1086888;
   t1[2085] := -0.0868463;
   t1[2086] := -0.043052;
   t1[2087] := -0.002035;
   t1[2088] := 0.034722;
   t1[2089] := 0.0663509;
   t1[2090] := 0.0922009;
   t1[2091] := 0.1116215;
   t1[2092] := 0.1239621;
   t1[2093] := 0.1285968;
   t1[2094] := 0.1261298;
   t1[2095] := 0.1189434;
   t1[2096] := 0.1095587;
   t1[2097] := 0.1004968;
   t1[2098] := 0.0942788;
   t1[2099] := 0.0929579;
   t1[2100] := 0.0361369;
   t1[2101] := 0.0184004;
   t1[2102] := -0.0031294;
   t1[2103] := -0.0285538;
   t1[2104] := -0.0559473;
   t1[2105] := -0.0826683;
   t1[2106] := -0.1060743;
   t1[2107] := -0.1235228;
   t1[2108] := -0.1324125;
   t1[2109] := -0.1322051;
   t1[2110] := -0.1253428;
   t1[2111] := -0.114501;
   t1[2112] := -0.102355;
   t1[2113] := -0.0915799;
   t1[2114] := -0.084454;
   t1[2115] := 0.1654816;
   t1[2116] := 0.1633248;
   t1[2117] := 0.1538973;
   t1[2118] := 0.1355376;
   t1[2119] := 0.1103259;
   t1[2120] := 0.0816646;
   t1[2121] := 0.0529576;
   t1[2122] := 0.027609;
   t1[2123] := 0.0089943;
   t1[2124] := -0.0009292;
   t1[2125] := -0.0022539;
   t1[2126] := 0.0047679;
   t1[2127] := 0.0198836;
   t1[2128] := 0.0428408;
   t1[2129] := 0.0730406;
   t1[2130] := 0.0828472;
   t1[2131] := 0.0479028;
   t1[2132] := 0.0097325;
   t1[2133] := -0.0303305;
   t1[2134] := -0.0694608;
   t1[2135] := -0.104306;
   t1[2136] := -0.1315129;
   t1[2137] := -0.1477285;
   t1[2138] := -0.1496556;
   t1[2139] := -0.1367942;
   t1[2140] := -0.1126867;
   t1[2141] := -0.0811913;
   t1[2142] := -0.0461659;
   t1[2143] := -0.0114688;
   t1[2144] := 0.0193897;
   t1[2145] := 0.0983107;
   t1[2146] := 0.0892271;
   t1[2147] := 0.0848777;
   t1[2148] := 0.0868591;
   t1[2149] := 0.0934296;
   t1[2150] := 0.1016686;
   t1[2151] := 0.1086537;
   t1[2152] := 0.111463;
   t1[2153] := 0.1072124;
   t1[2154] := 0.0949376;
   t1[2155] := 0.0764479;
   t1[2156] := 0.0537692;
   t1[2157] := 0.0289275;
   t1[2158] := 0.0039486;
   t1[2159] := -0.0193057;
   t1[2160] := 0.0484136;
   t1[2161] := 0.0314107;
   t1[2162] := 0.0156454;
   t1[2163] := 0.0035847;
   t1[2164] := -0.0047847;
   t1[2165] := -0.0103525;
   t1[2166] := -0.0140095;
   t1[2167] := -0.0166466;
   t1[2168] := -0.0191425;
   t1[2169] := -0.0217761;
   t1[2170] := -0.0239593;
   t1[2171] := -0.0250363;
   t1[2172] := -0.0243512;
   t1[2173] := -0.0212483;
   t1[2174] := -0.0151254;
   t1[2175] := 0.0102093;
   t1[2176] := 0.0401626;
   t1[2177] := 0.0657538;
   t1[2178] := 0.0834105;
   t1[2179] := 0.0935218;
   t1[2180] := 0.0978768;
   t1[2181] := 0.0982659;
   t1[2182] := 0.0964799;
   t1[2183] := 0.0942757;
   t1[2184] := 0.0917404;
   t1[2185] := 0.0865467;
   t1[2186] := 0.076179;
   t1[2187] := 0.0581217;
   t1[2188] := 0.0298591;
   t1[2189] := -0.0103927;
   t1[2190] := 0.0325954;
   t1[2191] := 0.0267495;
   t1[2192] := 0.023478;
   t1[2193] := 0.0234019;
   t1[2194] := 0.0265509;
   t1[2195] := 0.032746;
   t1[2196] := 0.0418081;
   t1[2197] := 0.053558;
   t1[2198] := 0.0678131;
   t1[2199] := 0.0842206;
   t1[2200] := 0.1021819;
   t1[2201] := 0.1210793;
   t1[2202] := 0.140295;
   t1[2203] := 0.1592113;
   t1[2204] := 0.1771791;
   t1[2205] := -0.0480857;
   t1[2206] := -0.0554614;
   t1[2207] := -0.0635384;
   t1[2208] := -0.0724774;
   t1[2209] := -0.0806222;
   t1[2210] := -0.0856748;
   t1[2211] := -0.0853362;
   t1[2212] := -0.0773075;
   t1[2213] := -0.0593425;
   t1[2214] := -0.0318256;
   t1[2215] := 0.001057;
   t1[2216] := 0.0348223;
   t1[2217] := 0.0649871;
   t1[2218] := 0.0870684;
   t1[2219] := 0.0972563;
   t1[2220] := 0.0970004;
   t1[2221] := 0.1142103;
   t1[2222] := 0.123124;
   t1[2223] := 0.1204171;
   t1[2224] := 0.1066652;
   t1[2225] := 0.0838219;
   t1[2226] := 0.0538422;
   t1[2227] := 0.0186813;
   t1[2228] := -0.0197008;
   t1[2229] := -0.0590968;
   t1[2230] := -0.0969423;
   t1[2231] := -0.1306447;
   t1[2232] := -0.1576117;
   t1[2233] := -0.1752509;
   t1[2234] := -0.1814605;
   t1[2235] := -0.0416155;
   t1[2236] := -0.0363205;
   t1[2237] := -0.0322986;
   t1[2238] := -0.0298126;
   t1[2239] := -0.0278406;
   t1[2240] := -0.0249069;
   t1[2241] := -0.0195352;
   t1[2242] := -0.0102493;
   t1[2243] := 0.0044049;
   t1[2244] := 0.0247709;
   t1[2245] := 0.0495871;
   t1[2246] := 0.0774666;
   t1[2247] := 0.1070226;
   t1[2248] := 0.1368683;
   t1[2249] := 0.1655431;
   t1[2250] := -0.3362626;
   t1[2251] := -0.3238524;
   t1[2252] := -0.2960049;
   t1[2253] := -0.2494259;
   t1[2254] := -0.1886314;
   t1[2255] := -0.1208974;
   t1[2256] := -0.0535033;
   t1[2257] := 0.0062719;
   t1[2258] := 0.0512357;
   t1[2259] := 0.0785333;
   t1[2260] := 0.0915789;
   t1[2261] := 0.0942763;
   t1[2262] := 0.0905289;
   t1[2263] := 0.0842406;
   t1[2264] := 0.078863;
   t1[2265] := -0.041304;
   t1[2266] := -0.0510186;
   t1[2267] := -0.0548829;
   t1[2268] := -0.0503896;
   t1[2269] := -0.0386208;
   t1[2270] := -0.0219271;
   t1[2271] := -0.0026607;
   t1[2272] := 0.0168265;
   t1[2273] := 0.0342119;
   t1[2274] := 0.0486465;
   t1[2275] := 0.0614107;
   t1[2276] := 0.0739514;
   t1[2277] := 0.0877154;
   t1[2278] := 0.1041494;
   t1[2279] := 0.124221;
   t1[2280] := -0.081103;
   t1[2281] := -0.0718181;
   t1[2282] := -0.0437795;
   t1[2283] := 0.0072145;
   t1[2284] := 0.074476;
   t1[2285] := 0.147469;
   t1[2286] := 0.2156533;
   t1[2287] := 0.2684888;
   t1[2288] := 0.2955715;
   t1[2289] := 0.2933263;
   t1[2290] := 0.268046;
   t1[2291] := 0.2267942;
   t1[2292] := 0.1766344;
   t1[2293] := 0.1246301;
   t1[2294] := 0.0772044;
   t1[2295] := -0.2409963;
   t1[2296] := -0.2126968;
   t1[2297] := -0.1793427;
   t1[2298] := -0.141921;
   t1[2299] := -0.1026364;
   t1[2300] := -0.0641238;
   t1[2301] := -0.0290186;
   t1[2302] := 4.39E-05;
   t1[2303] := 0.0204688;
   t1[2304] := 0.0316872;
   t1[2305] := 0.0360583;
   t1[2306] := 0.0361698;
   t1[2307] := 0.0346096;
   t1[2308] := 0.0339653;
   t1[2309] := 0.0364288;
   t1[2310] := -0.0666898;
   t1[2311] := -0.0113142;
   t1[2312] := 0.0338042;
   t1[2313] := 0.0640711;
   t1[2314] := 0.0806764;
   t1[2315] := 0.0868541;
   t1[2316] := 0.0858407;
   t1[2317] := 0.0808725;
   t1[2318] := 0.0751562;
   t1[2319] := 0.0704156;
   t1[2320] := 0.0662314;
   t1[2321] := 0.0620169;
   t1[2322] := 0.0571854;
   t1[2323] := 0.0511503;
   t1[2324] := 0.0434313;
   t1[2325] := 0.1049496;
   t1[2326] := 0.1323107;
   t1[2327] := 0.153373;
   t1[2328] := 0.1662057;
   t1[2329] := 0.1697528;
   t1[2330] := 0.1632669;
   t1[2331] := 0.1460012;
   t1[2332] := 0.1172088;
   t1[2333] := 0.0761932;
   t1[2334] := 0.0247878;
   t1[2335] := -0.0315181;
   t1[2336] := -0.0869497;
   t1[2337] := -0.1357323;
   t1[2338] := -0.1720912;
   t1[2339] := -0.1911876;
   t1[2340] := 0.1809488;
   t1[2341] := 0.1788293;
   t1[2342] := 0.1673001;
   t1[2343] := 0.1457947;
   t1[2344] := 0.1160177;
   t1[2345] := 0.0804761;
   t1[2346] := 0.0416781;
   t1[2347] := 0.0021314;
   t1[2348] := -0.0356707;
   t1[2349] := -0.0699813;
   t1[2350] := -0.1001317;
   t1[2351] := -0.1255373;
   t1[2352] := -0.1456136;
   t1[2353] := -0.159776;
   t1[2354] := -0.1675026;
   t1[2355] := -0.1985649;
   t1[2356] := -0.1789836;
   t1[2357] := -0.1483537;
   t1[2358] := -0.104728;
   t1[2359] := -0.0510856;
   t1[2360] := 0.0078536;
   t1[2361] := 0.0673682;
   t1[2362] := 0.1227364;
   t1[2363] := 0.1692733;
   t1[2364] := 0.2041326;
   t1[2365] := 0.2271252;
   t1[2366] := 0.2382695;
   t1[2367] := 0.2375839;
   t1[2368] := 0.2250868;
   t1[2369] := 0.2011627;
   t1[2370] := 0.1955927;
   t1[2371] := 0.1941393;
   t1[2372] := 0.1865643;
   t1[2373] := 0.1744535;
   t1[2374] := 0.1582534;
   t1[2375] := 0.1380075;
   t1[2376] := 0.1137588;
   t1[2377] := 0.0855505;
   t1[2378] := 0.0534454;
   t1[2379] := 0.0184971;
   t1[2380] := -0.0168092;
   t1[2381] := -0.0498764;
   t1[2382] := -0.0781074;
   t1[2383] := -0.0989054;
   t1[2384] := -0.1100764;
   t1[2385] := -0.1867194;
   t1[2386] := -0.1462405;
   t1[2387] := -0.0964243;
   t1[2388] := -0.0370777;
   t1[2389] := 0.0285334;
   t1[2390] := 0.0959202;
   t1[2391] := 0.1605929;
   t1[2392] := 0.2180612;
   t1[2393] := 0.2638592;
   t1[2394] := 0.2947079;
   t1[2395] := 0.309045;
   t1[2396] := 0.3054423;
   t1[2397] := 0.2824711;
   t1[2398] := 0.2387031;
   t1[2399] := 0.1737026;
   t1[2400] := 0.0990999;
   t1[2401] := 0.0827137;
   t1[2402] := 0.0686198;
   t1[2403] := 0.0577134;
   t1[2404] := 0.0495919;
   t1[2405] := 0.043394;
   t1[2406] := 0.038258;
   t1[2407] := 0.0333222;
   t1[2408] := 0.0277453;
   t1[2409] := 0.0217068;
   t1[2410] := 0.0168618;
   t1[2411] := 0.0149802;
   t1[2412] := 0.0178323;
   t1[2413] := 0.0271883;
   t1[2414] := 0.0442623;
   t1[2415] := 0.0896176;
   t1[2416] := 0.0780298;
   t1[2417] := 0.0622812;
   t1[2418] := 0.0413666;
   t1[2419] := 0.0168219;
   t1[2420] := -0.0089189;
   t1[2421] := -0.0334208;
   t1[2422] := -0.0542489;
   t1[2423] := -0.0689958;
   t1[2424] := -0.0766348;
   t1[2425] := -0.0781344;
   t1[2426] := -0.0746189;
   t1[2427] := -0.0672128;
   t1[2428] := -0.0570403;
   t1[2429] := -0.0452046;
   t1[2430] := 0.1495799;
   t1[2431] := 0.111068;
   t1[2432] := 0.0704512;
   t1[2433] := 0.0306892;
   t1[2434] := -0.0065241;
   t1[2435] := -0.0399419;
   t1[2436] := -0.0683179;
   t1[2437] := -0.0904059;
   t1[2438] := -0.1049763;
   t1[2439] := -0.1116388;
   t1[2440] := -0.1112155;
   t1[2441] := -0.1046234;
   t1[2442] := -0.0927793;
   t1[2443] := -0.0766002;
   t1[2444] := -0.0570968;
   t1[2445] := -0.0505247;
   t1[2446] := -0.0400901;
   t1[2447] := -0.0254102;
   t1[2448] := -0.0091421;
   t1[2449] := 0.0077119;
   t1[2450] := 0.024734;
   t1[2451] := 0.0415071;
   t1[2452] := 0.057614;
   t1[2453] := 0.0726383;
   t1[2454] := 0.0861988;
   t1[2455] := 0.0979656;
   t1[2456] := 0.1076123;
   t1[2457] := 0.1148129;
   t1[2458] := 0.1192412;
   t1[2459] := 0.1206185;
   t1[2460] := 0.0871255;
   t1[2461] := 0.0742433;
   t1[2462] := 0.060897;
   t1[2463] := 0.0494494;
   t1[2464] := 0.0399901;
   t1[2465] := 0.0318059;
   t1[2466] := 0.0241828;
   t1[2467] := 0.0164065;
   t1[2468] := 0.0077679;
   t1[2469] := -0.002188;
   t1[2470] := -0.0135494;
   t1[2471] := -0.0263758;
   t1[2472] := -0.0407265;
   t1[2473] := -0.056661;
   t1[2474] := -0.07405;
   t1[2475] := -0.0546469;
   t1[2476] := -0.0991847;
   t1[2477] := -0.133845;
   t1[2478] := -0.1548857;
   t1[2479] := -0.1628136;
   t1[2480] := -0.1596361;
   t1[2481] := -0.1473626;
   t1[2482] := -0.1280025;
   t1[2483] := -0.1035689;
   t1[2484] := -0.0762694;
   t1[2485] := -0.0485923;
   t1[2486] := -0.0230479;
   t1[2487] := -0.0021463;
   t1[2488] := 0.0116022;
   t1[2489] := 0.0161952;
   t1[2490] := -0.0097633;
   t1[2491] := 0.0035987;
   t1[2492] := 0.0172484;
   t1[2493] := 0.029957;
   t1[2494] := 0.0411298;
   t1[2495] := 0.0503968;
   t1[2496] := 0.0573877;
   t1[2497] := 0.0617325;
   t1[2498] := 0.0630718;
   t1[2499] := 0.0615695;
   t1[2500] := 0.0581464;
   t1[2501] := 0.0537823;
   t1[2502] := 0.0494569;
   t1[2503] := 0.0461503;
   t1[2504] := 0.0446689;
   t1[2505] := 0.4198114;
   t1[2506] := 0.3935941;
   t1[2507] := 0.3487166;
   t1[2508] := 0.2835445;
   t1[2509] := 0.2037699;
   t1[2510] := 0.117674;
   t1[2511] := 0.0335407;
   t1[2512] := -0.040346;
   t1[2513] := -0.0958;
   t1[2514] := -0.1295343;
   t1[2515] := -0.145342;
   t1[2516] := -0.147569;
   t1[2517] := -0.1405613;
   t1[2518] := -0.1286646;
   t1[2519] := -0.1158025;
   t1[2520] := 0.0019711;
   t1[2521] := 0.0022643;
   t1[2522] := 0.0058747;
   t1[2523] := 0.0132652;
   t1[2524] := 0.0249988;
   t1[2525] := 0.0416735;
   t1[2526] := 0.0638875;
   t1[2527] := 0.0922389;
   t1[2528] := 0.1272807;
   t1[2529] := 0.167303;
   t1[2530] := 0.2073259;
   t1[2531] := 0.2421143;
   t1[2532] := 0.2664329;
   t1[2533] := 0.2750465;
   t1[2534] := 0.2637612;
   t1[2535] := -0.0018019;
   t1[2536] := 0.0146538;
   t1[2537] := 0.0305786;
   t1[2538] := 0.0444612;
   t1[2539] := 0.0564392;
   t1[2540] := 0.0672328;
   t1[2541] := 0.077563;
   t1[2542] := 0.0881508;
   t1[2543] := 0.0996916;
   t1[2544] := 0.1116036;
   t1[2545] := 0.1214594;
   t1[2546] := 0.1266872;
   t1[2547] := 0.1247156;
   t1[2548] := 0.1129728;
   t1[2549] := 0.0895944;
   t1[2550] := 0.046532;
   t1[2551] := 0.0740913;
   t1[2552] := 0.0924658;
   t1[2553] := 0.0974729;
   t1[2554] := 0.0911579;
   t1[2555] := 0.0777667;
   t1[2556] := 0.0615478;
   t1[2557] := 0.0467495;
   t1[2558] := 0.037565;
   t1[2559] := 0.035419;
   t1[2560] := 0.0377355;
   t1[2561] := 0.0416258;
   t1[2562] := 0.0442017;
   t1[2563] := 0.0425747;
   t1[2564] := 0.0343558;
   t1[2565] := 0.1429637;
   t1[2566] := 0.1522729;
   t1[2567] := 0.1561933;
   t1[2568] := 0.153325;
   t1[2569] := 0.1450948;
   t1[2570] := 0.1339282;
   t1[2571] := 0.1222518;
   t1[2572] := 0.1124922;
   t1[2573] := 0.1070483;
   t1[2574] := 0.1069224;
   t1[2575] := 0.1110987;
   t1[2576] := 0.1184043;
   t1[2577] := 0.1276658;
   t1[2578] := 0.13771;
   t1[2579] := 0.1474286;
   t1[2580] := 0.1319272;
   t1[2581] := 0.1650362;
   t1[2582] := 0.196325;
   t1[2583] := 0.2229424;
   t1[2584] := 0.2431984;
   t1[2585] := 0.2558133;
   t1[2586] := 0.2595075;
   t1[2587] := 0.2530018;
   t1[2588] := 0.235046;
   t1[2589] := 0.205849;
   t1[2590] := 0.1677283;
   t1[2591] := 0.1231661;
   t1[2592] := 0.0746446;
   t1[2593] := 0.024646;
   t1[2594] := -0.0245742;
   t1[2595] := 0.2096563;
   t1[2596] := 0.2054805;
   t1[2597] := 0.1987581;
   t1[2598] := 0.1897786;
   t1[2599] := 0.179163;
   t1[2600] := 0.16765;
   t1[2601] := 0.1559782;
   t1[2602] := 0.1448863;
   t1[2603] := 0.1351162;
   t1[2604] := 0.1275734;
   t1[2605] := 0.1233993;
   t1[2606] := 0.1237541;
   t1[2607] := 0.1297977;
   t1[2608] := 0.1426901;
   t1[2609] := 0.1631009;
   t1[2610] := 0.1127695;
   t1[2611] := 0.1185965;
   t1[2612] := 0.1269101;
   t1[2613] := 0.1380314;
   t1[2614] := 0.1501462;
   t1[2615] := 0.1606855;
   t1[2616] := 0.1670797;
   t1[2617] := 0.1667594;
   t1[2618] := 0.1571921;
   t1[2619] := 0.1377146;
   t1[2620] := 0.1103647;
   t1[2621] := 0.077391;
   t1[2622] := 0.0410421;
   t1[2623] := 0.0035668;
   t1[2624] := -0.0328668;
   t1[2625] := 0.1020229;
   t1[2626] := 0.1037319;
   t1[2627] := 0.10323;
   t1[2628] := 0.0999524;
   t1[2629] := 0.0943676;
   t1[2630] := 0.087309;
   t1[2631] := 0.0796109;
   t1[2632] := 0.0721071;
   t1[2633] := 0.0656238;
   t1[2634] := 0.0605871;
   t1[2635] := 0.0568448;
   t1[2636] := 0.0542001;
   t1[2637] := 0.0524558;
   t1[2638] := 0.0514148;
   t1[2639] := 0.0508935;
   t1[2640] := 0.0456957;
   t1[2641] := 0.0505849;
   t1[2642] := 0.0568825;
   t1[2643] := 0.0629849;
   t1[2644] := 0.0691703;
   t1[2645] := 0.0763821;
   t1[2646] := 0.0855644;
   t1[2647] := 0.0976612;
   t1[2648] := 0.1135942;
   t1[2649] := 0.1331585;
   t1[2650] := 0.154521;
   t1[2651] := 0.1757216;
   t1[2652] := 0.1948002;
   t1[2653] := 0.2097967;
   t1[2654] := 0.2189999;
   t1[2655] := 0.0563676;
   t1[2656] := 0.030645;
   t1[2657] := 0.0133273;
   t1[2658] := 0.0074349;
   t1[2659] := 0.011341;
   t1[2660] := 0.0217775;
   t1[2661] := 0.0354739;
   t1[2662] := 0.04916;
   t1[2663] := 0.0596003;
   t1[2664] := 0.0652992;
   t1[2665] := 0.0672756;
   t1[2666] := 0.0667448;
   t1[2667] := 0.0649221;
   t1[2668] := 0.0630227;
   t1[2669] := 0.0620756;
   t1[2670] := -0.0260615;
   t1[2671] := -0.0042681;
   t1[2672] := 0.0150406;
   t1[2673] := 0.0311598;
   t1[2674] := 0.0437835;
   t1[2675] := 0.0527461;
   t1[2676] := 0.0578824;
   t1[2677] := 0.0590271;
   t1[2678] := 0.0560231;
   t1[2679] := 0.0491177;
   t1[2680] := 0.0391433;
   t1[2681] := 0.0269779;
   t1[2682] := 0.0134995;
   t1[2683] := -0.0004139;
   t1[2684] := -0.0138996;
   t1[2685] := 0.1002057;
   t1[2686] := 0.1034546;
   t1[2687] := 0.1115845;
   t1[2688] := 0.1246809;
   t1[2689] := 0.1404212;
   t1[2690] := 0.1556314;
   t1[2691] := 0.1671365;
   t1[2692] := 0.1717619;
   t1[2693] := 0.1663827;
   t1[2694] := 0.1503928;
   t1[2695] := 0.1268251;
   t1[2696] := 0.0989966;
   t1[2697] := 0.0702245;
   t1[2698] := 0.0438258;
   t1[2699] := 0.0226909;
   t1[2700] := 0.2653609;
   t1[2701] := 0.2587946;
   t1[2702] := 0.2512794;
   t1[2703] := 0.2427861;
   t1[2704] := 0.2327362;
   t1[2705] := 0.2203571;
   t1[2706] := 0.2048762;
   t1[2707] := 0.1855208;
   t1[2708] := 0.1615378;
   t1[2709] := 0.1331538;
   t1[2710] := 0.1020116;
   t1[2711] := 0.0698644;
   t1[2712] := 0.0384655;
   t1[2713] := 0.009568;
   t1[2714] := -0.0152517;
   t1[2715] := 0.1547851;
   t1[2716] := 0.1564473;
   t1[2717] := 0.1597121;
   t1[2718] := 0.1639812;
   t1[2719] := 0.1679386;
   t1[2720] := 0.1700145;
   t1[2721] := 0.1686388;
   t1[2722] := 0.1622413;
   t1[2723] := 0.1492919;
   t1[2724] := 0.1302518;
   t1[2725] := 0.1084608;
   t1[2726] := 0.0874832;
   t1[2727] := 0.0708833;
   t1[2728] := 0.0622256;
   t1[2729] := 0.064316;
   t1[2730] := 0.2072259;
   t1[2731] := 0.1901705;
   t1[2732] := 0.1720155;
   t1[2733] := 0.1544939;
   t1[2734] := 0.139005;
   t1[2735] := 0.1268307;
   t1[2736] := 0.1192524;
   t1[2737] := 0.1175517;
   t1[2738] := 0.122971;
   t1[2739] := 0.1347973;
   t1[2740] := 0.1494914;
   t1[2741] := 0.1632937;
   t1[2742] := 0.1724445;
   t1[2743] := 0.1731839;
   t1[2744] := 0.1624853;
   t1[2745] := 0.2724063;
   t1[2746] := 0.2428027;
   t1[2747] := 0.2122088;
   t1[2748] := 0.1828237;
   t1[2749] := 0.1545416;
   t1[2750] := 0.1264418;
   t1[2751] := 0.0976031;
   t1[2752] := 0.0671039;
   t1[2753] := 0.0340323;
   t1[2754] := -0.0020565;
   t1[2755] := -0.0409316;
   t1[2756] := -0.0823095;
   t1[2757] := -0.1259065;
   t1[2758] := -0.1714393;
   t1[2759] := -0.2182391;
   t1[2760] := 0.1602175;
   t1[2761] := 0.1784402;
   t1[2762] := 0.1963308;
   t1[2763] := 0.2125517;
   t1[2764] := 0.2261795;
   t1[2765] := 0.2364367;
   t1[2766] := 0.242546;
   t1[2767] := 0.2437301;
   t1[2768] := 0.2392264;
   t1[2769] := 0.2290019;
   t1[2770] := 0.2140784;
   t1[2771] := 0.1955599;
   t1[2772] := 0.1745504;
   t1[2773] := 0.1521539;
   t1[2774] := 0.1294562;
   t1[2775] := 0.120246;
   t1[2776] := 0.1217794;
   t1[2777] := 0.1214958;
   t1[2778] := 0.1206101;
   t1[2779] := 0.1195939;
   t1[2780] := 0.1186561;
   t1[2781] := 0.1180055;
   t1[2782] := 0.1178506;
   t1[2783] := 0.1184055;
   t1[2784] := 0.1201516;
   t1[2785] := 0.1239572;
   t1[2786] := 0.1307206;
   t1[2787] := 0.1413403;
   t1[2788] := 0.1567145;
   t1[2789] := 0.1772589;
   t1[2790] := 0.0852868;
   t1[2791] := 0.0824586;
   t1[2792] := 0.0844848;
   t1[2793] := 0.0911939;
   t1[2794] := 0.1011767;
   t1[2795] := 0.1125869;
   t1[2796] := 0.1235776;
   t1[2797] := 0.1323019;
   t1[2798] := 0.1369372;
   t1[2799] := 0.1368771;
   t1[2800] := 0.133272;
   t1[2801] := 0.1274098;
   t1[2802] := 0.1205784;
   t1[2803] := 0.1140657;
   t1[2804] := 0.1089268;
   t1[2805] := 0.2002328;
   t1[2806] := 0.2033647;
   t1[2807] := 0.1975502;
   t1[2808] := 0.1792453;
   t1[2809] := 0.1492452;
   t1[2810] := 0.1098784;
   t1[2811] := 0.0634749;
   t1[2812] := 0.0123651;
   t1[2813] := -0.0411058;
   t1[2814] := -0.0938431;
   t1[2815] := -0.1416683;
   t1[2816] := -0.1803185;
   t1[2817] := -0.2055308;
   t1[2818] := -0.2130424;
   t1[2819] := -0.1996302;
   t1[2820] := -0.0673173;
   t1[2821] := -0.0611401;
   t1[2822] := -0.0474342;
   t1[2823] := -0.0241686;
   t1[2824] := 0.0069945;
   t1[2825] := 0.0430876;
   t1[2826] := 0.0811421;
   t1[2827] := 0.1181893;
   t1[2828] := 0.1512851;
   t1[2829] := 0.1787289;
   t1[2830] := 0.2006162;
   t1[2831] := 0.2171832;
   t1[2832] := 0.2286658;
   t1[2833] := 0.2353;
   t1[2834] := 0.2372926;
   t1[2835] := 0.1328057;
   t1[2836] := 0.1341211;
   t1[2837] := 0.1272074;
   t1[2838] := 0.1122947;
   t1[2839] := 0.0909306;
   t1[2840] := 0.0651283;
   t1[2841] := 0.0369014;
   t1[2842] := 0.0082635;
   t1[2843] := -0.0187797;
   t1[2844] := -0.0426151;
   t1[2845] := -0.0621975;
   t1[2846] := -0.076526;
   t1[2847] := -0.0845998;
   t1[2848] := -0.0854179;
   t1[2849] := -0.0783289;
   t1[2850] := -0.0581343;
   t1[2851] := -0.0133043;
   t1[2852] := 0.0309237;
   t1[2853] := 0.0718275;
   t1[2854] := 0.1081703;
   t1[2855] := 0.1392398;
   t1[2856] := 0.1643245;
   t1[2857] := 0.1827127;
   t1[2858] := 0.1937057;
   t1[2859] := 0.1972426;
   t1[2860] := 0.1941846;
   t1[2861] := 0.1854647;
   t1[2862] := 0.1720163;
   t1[2863] := 0.1547723;
   t1[2864] := 0.1346985;
   t1[2865] := 0.0822117;
   t1[2866] := 0.0790527;
   t1[2867] := 0.0802027;
   t1[2868] := 0.0889129;
   t1[2869] := 0.1022555;
   t1[2870] := 0.1151196;
   t1[2871] := 0.1223914;
   t1[2872] := 0.1189574;
   t1[2873] := 0.0998009;
   t1[2874] := 0.0647515;
   t1[2875] := 0.020643;
   t1[2876] := -0.0251438;
   t1[2877] := -0.0652283;
   t1[2878] := -0.09223;
   t1[2879] := -0.1000393;
   t1[2880] := 0.0261083;
   t1[2881] := 0.0255114;
   t1[2882] := 0.0301572;
   t1[2883] := 0.0414563;
   t1[2884] := 0.0584277;
   t1[2885] := 0.079245;
   t1[2886] := 0.1020806;
   t1[2887] := 0.1251073;
   t1[2888] := 0.1465082;
   t1[2889] := 0.1649886;
   t1[2890] := 0.1800087;
   t1[2891] := 0.1910877;
   t1[2892] := 0.1977448;
   t1[2893] := 0.1994991;
   t1[2894] := 0.1960069;
   t1[2895] := 0.0666804;
   t1[2896] := 0.0504849;
   t1[2897] := 0.0383564;
   t1[2898] := 0.0348998;
   t1[2899] := 0.0390518;
   t1[2900] := 0.0477465;
   t1[2901] := 0.0579156;
   t1[2902] := 0.066491;
   t1[2903] := 0.0704401;
   t1[2904] := 0.0685266;
   t1[2905] := 0.0621092;
   t1[2906] := 0.0527495;
   t1[2907] := 0.0420089;
   t1[2908] := 0.031449;
   t1[2909] := 0.0224616;
   t1[2910] := 0.032325;
   t1[2911] := 0.0350114;
   t1[2912] := 0.0424177;
   t1[2913] := 0.0557425;
   t1[2914] := 0.0736159;
   t1[2915] := 0.0937606;
   t1[2916] := 0.1138978;
   t1[2917] := 0.1317492;
   t1[2918] := 0.1450601;
   t1[2919] := 0.1527777;
   t1[2920] := 0.1555859;
   t1[2921] := 0.154304;
   t1[2922] := 0.1497514;
   t1[2923] := 0.1427476;
   t1[2924] := 0.1340508;
   t1[2925] := -0.0474794;
   t1[2926] := -0.0473073;
   t1[2927] := -0.0410615;
   t1[2928] := -0.0261021;
   t1[2929] := -0.0035912;
   t1[2930] := 0.0239656;
   t1[2931] := 0.0540613;
   t1[2932] := 0.0841888;
   t1[2933] := 0.1118543;
   t1[2934] := 0.1352315;
   t1[2935] := 0.1534585;
   t1[2936] := 0.1657489;
   t1[2937] := 0.1713161;
   t1[2938] := 0.1693738;
   t1[2939] := 0.1594401;
   t1[2940] := -0.1618689;
   t1[2941] := -0.1203332;
   t1[2942] := -0.0792785;
   t1[2943] := -0.0414959;
   t1[2944] := -0.0078523;
   t1[2945] := 0.0214649;
   t1[2946] := 0.046269;
   t1[2947] := 0.0663734;
   t1[2948] := 0.0815918;
   t1[2949] := 0.0917562;
   t1[2950] := 0.0967242;
   t1[2951] := 0.0963559;
   t1[2952] := 0.0905111;
   t1[2953] := 0.0790498;
   t1[2954] := 0.0620609;
   t1[2955] := -0.108307;
   t1[2956] := -0.0982721;
   t1[2957] := -0.0845619;
   t1[2958] := -0.0666727;
   t1[2959] := -0.0453051;
   t1[2960] := -0.021585;
   t1[2961] := 0.003361;
   t1[2962] := 0.0284065;
   t1[2963] := 0.0524334;
   t1[2964] := 0.074749;
   t1[2965] := 0.0952747;
   t1[2966] := 0.11398;
   t1[2967] := 0.1308344;
   t1[2968] := 0.1458075;
   t1[2969] := 0.158707;
   t1[2970] := -0.0744484;
   t1[2971] := -0.0611159;
   t1[2972] := -0.0407944;
   t1[2973] := -0.0119923;
   t1[2974] := 0.023732;
   t1[2975] := 0.0637421;
   t1[2976] := 0.1054004;
   t1[2977] := 0.1460696;
   t1[2978] := 0.1831266;
   t1[2979] := 0.214675;
   t1[2980] := 0.239868;
   t1[2981] := 0.2579411;
   t1[2982] := 0.2681296;
   t1[2983] := 0.2696691;
   t1[2984] := 0.2620204;
   t1[2985] := 0.147486;
   t1[2986] := 0.1326573;
   t1[2987] := 0.111248;
   t1[2988] := 0.083335;
   t1[2989] := 0.0509007;
   t1[2990] := 0.0166008;
   t1[2991] := -0.0169079;
   t1[2992] := -0.046969;
   t1[2993] := -0.0709583;
   t1[2994] := -0.0878764;
   t1[2995] := -0.0990721;
   t1[2996] := -0.1060772;
   t1[2997] := -0.1104238;
   t1[2998] := -0.1136438;
   t1[2999] := -0.1170604;
   t1[3000] := -0.1079736;
   t1[3001] := -0.0849456;
   t1[3002] := -0.0556524;
   t1[3003] := -0.0215777;
   t1[3004] := 0.0142717;
   t1[3005] := 0.0483511;
   t1[3006] := 0.0771147;
   t1[3007] := 0.0970171;
   t1[3008] := 0.1045737;
   t1[3009] := 0.0993471;
   t1[3010] := 0.0853035;
   t1[3011] := 0.0667533;
   t1[3012] := 0.0480066;
   t1[3013] := 0.0333737;
   t1[3014] := 0.0263849;
   t1[3015] := 0.2213627;
   t1[3016] := 0.2036206;
   t1[3017] := 0.1822179;
   t1[3018] := 0.1589792;
   t1[3019] := 0.1343747;
   t1[3020] := 0.1083963;
   t1[3021] := 0.0810352;
   t1[3022] := 0.0522827;
   t1[3023] := 0.0221504;
   t1[3024] := -0.0083273;
   t1[3025] := -0.036638;
   t1[3026] := -0.0601539;
   t1[3027] := -0.0762473;
   t1[3028] := -0.0822904;
   t1[3029] := -0.0762452;
   t1[3030] := -0.0309151;
   t1[3031] := -0.0182399;
   t1[3032] := -0.004385;
   t1[3033] := 0.0098028;
   t1[3034] := 0.0247684;
   t1[3035] := 0.0414129;
   t1[3036] := 0.0606381;
   t1[3037] := 0.0833457;
   t1[3038] := 0.1104156;
   t1[3039] := 0.1416218;
   t1[3040] := 0.1751408;
   t1[3041] := 0.2090246;
   t1[3042] := 0.2413248;
   t1[3043] := 0.2700933;
   t1[3044] := 0.2935205;
   t1[3045] := 0.2227261;
   t1[3046] := 0.2374933;
   t1[3047] := 0.246712;
   t1[3048] := 0.2492314;
   t1[3049] := 0.2451685;
   t1[3050] := 0.235088;
   t1[3051] := 0.2195551;
   t1[3052] := 0.1991351;
   t1[3053] := 0.1744086;
   t1[3054] := 0.1467174;
   t1[3055] := 0.1185042;
   t1[3056] := 0.0922976;
   t1[3057] := 0.0706259;
   t1[3058] := 0.0560178;
   t1[3059] := 0.0505837;
   t1[3060] := -0.1056972;
   t1[3061] := -0.0901565;
   t1[3062] := -0.0754007;
   t1[3063] := -0.0622195;
   t1[3064] := -0.0494215;
   t1[3065] := -0.0351154;
   t1[3066] := -0.0174091;
   t1[3067] := 0.0055897;
   t1[3068] := 0.0357221;
   t1[3069] := 0.0722802;
   t1[3070] := 0.1108718;
   t1[3071] := 0.1468171;
   t1[3072] := 0.1754365;
   t1[3073] := 0.1920503;
   t1[3074] := 0.1928305;
   t1[3075] := 0.0595173;
   t1[3076] := 0.0844017;
   t1[3077] := 0.1010478;
   t1[3078] := 0.107219;
   t1[3079] := 0.1048149;
   t1[3080] := 0.0971966;
   t1[3081] := 0.0877268;
   t1[3082] := 0.0797683;
   t1[3083] := 0.0766259;
   t1[3084] := 0.078705;
   t1[3085] := 0.0822208;
   t1[3086] := 0.0830613;
   t1[3087] := 0.0771146;
   t1[3088] := 0.0602687;
   t1[3089] := 0.0293821;
   t1[3090] := 0.2665905;
   t1[3091] := 0.2140689;
   t1[3092] := 0.1633811;
   t1[3093] := 0.1208088;
   t1[3094] := 0.0874285;
   t1[3095] := 0.062477;
   t1[3096] := 0.0451894;
   t1[3097] := 0.0348005;
   t1[3098] := 0.0305435;
   t1[3099] := 0.0315676;
   t1[3100] := 0.0369006;
   t1[3101] := 0.0455608;
   t1[3102] := 0.0565664;
   t1[3103] := 0.0689358;
   t1[3104] := 0.0816562;
   t1[3105] := 0.1867516;
   t1[3106] := 0.2056049;
   t1[3107] := 0.2082826;
   t1[3108] := 0.1913536;
   t1[3109] := 0.1581045;
   t1[3110] := 0.1141964;
   t1[3111] := 0.0652925;
   t1[3112] := 0.0170565;
   t1[3113] := -0.0248979;
   t1[3114] := -0.0574399;
   t1[3115] := -0.0810277;
   t1[3116] := -0.0963996;
   t1[3117] := -0.1042941;
   t1[3118] := -0.1054494;
   t1[3119] := -0.1006877;
   t1[3120] := -0.1450596;
   t1[3121] := -0.1306753;
   t1[3122] := -0.1155462;
   t1[3123] := -0.1003355;
   t1[3124] := -0.0846022;
   t1[3125] := -0.0675154;
   t1[3126] := -0.0482434;
   t1[3127] := -0.0259549;
   t1[3128] := 0.000164;
   t1[3129] := 0.030041;
   t1[3130] := 0.0623233;
   t1[3131] := 0.0955581;
   t1[3132] := 0.1282926;
   t1[3133] := 0.159074;
   t1[3134] := 0.1864619;
   t1[3135] := 0.1540427;
   t1[3136] := 0.1530604;
   t1[3137] := 0.1491994;
   t1[3138] := 0.1435257;
   t1[3139] := 0.1359963;
   t1[3140] := 0.1261759;
   t1[3141] := 0.1136291;
   t1[3142] := 0.0979206;
   t1[3143] := 0.0786367;
   t1[3144] := 0.0564646;
   t1[3145] := 0.0336821;
   t1[3146] := 0.0126911;
   t1[3147] := -0.0041065;
   t1[3148] := -0.0143088;
   t1[3149] := -0.0160749;
   t1[3150] := 0.1028241;
   t1[3151] := 0.0938343;
   t1[3152] := 0.0854728;
   t1[3153] := 0.0782067;
   t1[3154] := 0.0719553;
   t1[3155] := 0.0664446;
   t1[3156] := 0.0614003;
   t1[3157] := 0.0565481;
   t1[3158] := 0.0516048;
   t1[3159] := 0.04584;
   t1[3160] := 0.0378774;
   t1[3161] := 0.02629;
   t1[3162] := 0.0096508;
   t1[3163] := -0.013467;
   t1[3164] := -0.0439089;
   t1[3165] := -0.2808648;
   t1[3166] := -0.2451323;
   t1[3167] := -0.2057925;
   t1[3168] := -0.1654068;
   t1[3169] := -0.1241551;
   t1[3170] := -0.0813762;
   t1[3171] := -0.0364076;
   t1[3172] := 0.0114131;
   t1[3173] := 0.0627152;
   t1[3174] := 0.1164765;
   t1[3175] := 0.1692878;
   t1[3176] := 0.2175535;
   t1[3177] := 0.2576782;
   t1[3178] := 0.2860665;
   t1[3179] := 0.2997592;
   t1[3180] := -0.2673689;
   t1[3181] := -0.2250907;
   t1[3182] := -0.1778593;
   t1[3183] := -0.1287648;
   t1[3184] := -0.0784491;
   t1[3185] := -0.0266891;
   t1[3186] := 0.0267391;
   t1[3187] := 0.0820597;
   t1[3188] := 0.1394509;
   t1[3189] := 0.1967915;
   t1[3190] := 0.2486379;
   t1[3191] := 0.2892871;
   t1[3192] := 0.3130357;
   t1[3193] := 0.3141808;
   t1[3194] := 0.2884052;
   t1[3195] := 0.2621492;
   t1[3196] := 0.2234307;
   t1[3197] := 0.1780936;
   t1[3198] := 0.1284713;
   t1[3199] := 0.0772303;
   t1[3200] := 0.0271545;
   t1[3201] := -0.0189719;
   t1[3202] := -0.0583647;
   t1[3203] := -0.0882735;
   t1[3204] := -0.1076462;
   t1[3205] := -0.1178839;
   t1[3206] := -0.1205798;
   t1[3207] := -0.1173268;
   t1[3208] := -0.1097179;
   t1[3209] := -0.0992634;
   t1[3210] := -0.0762902;
   t1[3211] := -0.0590757;
   t1[3212] := -0.0378554;
   t1[3213] := -0.0117545;
   t1[3214] := 0.0179102;
   t1[3215] := 0.0490478;
   t1[3216] := 0.0795666;
   t1[3217] := 0.1073747;
   t1[3218] := 0.1303934;
   t1[3219] := 0.1472086;
   t1[3220] := 0.1573657;
   t1[3221] := 0.1604855;
   t1[3222] := 0.1561886;
   t1[3223] := 0.1440954;
   t1[3224] := 0.1241142;
   t1[3225] := -0.2361995;
   t1[3226] := -0.2461585;
   t1[3227] := -0.2417233;
   t1[3228] := -0.2190281;
   t1[3229] := -0.180726;
   t1[3230] := -0.1317741;
   t1[3231] := -0.0771316;
   t1[3232] := -0.0217583;
   t1[3233] := 0.0294164;
   t1[3234] := 0.07296;
   t1[3235] := 0.1076036;
   t1[3236] := 0.1322475;
   t1[3237] := 0.1457915;
   t1[3238] := 0.1471359;
   t1[3239] := 0.1357482;
   t1[3240] := 0.2855396;
   t1[3241] := 0.2357897;
   t1[3242] := 0.1833328;
   t1[3243] := 0.131762;
   t1[3244] := 0.0816169;
   t1[3245] := 0.0323581;
   t1[3246] := -0.016555;
   t1[3247] := -0.0656631;
   t1[3248] := -0.1154763;
   t1[3249] := -0.1649826;
   t1[3250] := -0.2109701;
   t1[3251] := -0.2500551;
   t1[3252] := -0.278854;
   t1[3253] := -0.2939831;
   t1[3254] := -0.2927593;
   t1[3255] := 0.0307899;
   t1[3256] := 0.033017;
   t1[3257] := 0.0334862;
   t1[3258] := 0.0320249;
   t1[3259] := 0.0282673;
   t1[3260] := 0.0217793;
   t1[3261] := 0.0121266;
   t1[3262] := -0.001125;
   t1[3263] := -0.0183803;
   t1[3264] := -0.0385733;
   t1[3265] := -0.0585121;
   t1[3266] := -0.074839;
   t1[3267] := -0.084196;
   t1[3268] := -0.0832254;
   t1[3269] := -0.0693698;
   t1[3270] := 0.0672795;
   t1[3271] := 0.0337566;
   t1[3272] := 0.0102953;
   t1[3273] := -0.0001791;
   t1[3274] := 0.0001911;
   t1[3275] := 0.007473;
   t1[3276] := 0.0177316;
   t1[3277] := 0.027032;
   t1[3278] := 0.0314832;
   t1[3279] := 0.0293945;
   t1[3280] := 0.0222551;
   t1[3281] := 0.0118025;
   t1[3282] := -0.0002258;
   t1[3283] := -0.0120924;
   t1[3284] := -0.0222223;
   t1[3285] := 0.1889521;
   t1[3286] := 0.1266015;
   t1[3287] := 0.0663512;
   t1[3288] := 0.012052;
   t1[3289] := -0.0356978;
   t1[3290] := -0.0774491;
   t1[3291] := -0.113754;
   t1[3292] := -0.1451648;
   t1[3293] := -0.1722277;
   t1[3294] := -0.1951898;
   t1[3295] := -0.2138652;
   t1[3296] := -0.2280348;
   t1[3297] := -0.2374789;
   t1[3298] := -0.2419784;
   t1[3299] := -0.2413561;
   t1[3300] := 0.1528176;
   t1[3301] := 0.1173664;
   t1[3302] := 0.0844603;
   t1[3303] := 0.0560332;
   t1[3304] := 0.0324174;
   t1[3305] := 0.0133794;
   t1[3306] := -0.0013151;
   t1[3307] := -0.0119003;
   t1[3308] := -0.0186164;
   t1[3309] := -0.0219996;
   t1[3310] := -0.0230138;
   t1[3311] := -0.0226563;
   t1[3312] := -0.0219245;
   t1[3313] := -0.0218157;
   t1[3314] := -0.0231565;
   t1[3315] := 0.2206065;
   t1[3316] := 0.1527838;
   t1[3317] := 0.0971946;
   t1[3318] := 0.0610706;
   t1[3319] := 0.0409795;
   t1[3320] := 0.0297203;
   t1[3321] := 0.0200878;
   t1[3322] := 0.0048768;
   t1[3323] := -0.0230039;
   t1[3324] := -0.0649461;
   t1[3325] := -0.1141045;
   t1[3326] := -0.1629911;
   t1[3327] := -0.2041173;
   t1[3328] := -0.2299951;
   t1[3329] := -0.2344296;
   t1[3330] := 0.1708361;
   t1[3331] := 0.1505133;
   t1[3332] := 0.1257442;
   t1[3333] := 0.0975643;
   t1[3334] := 0.0671807;
   t1[3335] := 0.0358615;
   t1[3336] := 0.0048745;
   t1[3337] := -0.0245121;
   t1[3338] := -0.0510341;
   t1[3339] := -0.0736113;
   t1[3340] := -0.0914293;
   t1[3341] := -0.1036946;
   t1[3342] := -0.1096137;
   t1[3343] := -0.1083932;
   t1[3344] := -0.0995559;
   t1[3345] := -0.2305381;
   t1[3346] := -0.1919115;
   t1[3347] := -0.1474767;
   t1[3348] := -0.0979882;
   t1[3349] := -0.0452096;
   t1[3350] := 0.0087387;
   t1[3351] := 0.061736;
   t1[3352] := 0.1116615;
   t1[3353] := 0.156405;
   t1[3354] := 0.1943914;
   t1[3355] := 0.224818;
   t1[3356] := 0.2469425;
   t1[3357] := 0.2600229;
   t1[3358] := 0.2633169;
   t1[3359] := 0.2563623;
   t1[3360] := -0.0753599;
   t1[3361] := -0.0882749;
   t1[3362] := -0.098825;
   t1[3363] := -0.1065015;
   t1[3364] := -0.1095981;
   t1[3365] := -0.1059849;
   t1[3366] := -0.0935313;
   t1[3367] := -0.0701073;
   t1[3368] := -0.0336468;
   t1[3369] := 0.0146871;
   t1[3370] := 0.069065;
   t1[3371] := 0.1232933;
   t1[3372] := 0.1711782;
   t1[3373] := 0.2065262;
   t1[3374] := 0.2240977;
   t1[3375] := -0.0575768;
   t1[3376] := -0.0542202;
   t1[3377] := -0.0482553;
   t1[3378] := -0.0393255;
   t1[3379] := -0.0268107;
   t1[3380] := -0.0099981;
   t1[3381] := 0.0118254;
   t1[3382] := 0.0393729;
   t1[3383] := 0.0733054;
   t1[3384] := 0.111674;
   t1[3385] := 0.1487579;
   t1[3386] := 0.1785422;
   t1[3387] := 0.1950117;
   t1[3388] := 0.1921513;
   t1[3389] := 0.1654336;
   t1[3390] := 0.0130781;
   t1[3391] := 0.0115276;
   t1[3392] := 0.0140124;
   t1[3393] := 0.021848;
   t1[3394] := 0.0337342;
   t1[3395] := 0.0474469;
   t1[3396] := 0.0607606;
   t1[3397] := 0.0714501;
   t1[3398] := 0.0773152;
   t1[3399] := 0.0774254;
   t1[3400] := 0.0726838;
   t1[3401] := 0.0641371;
   t1[3402] := 0.052832;
   t1[3403] := 0.0398148;
   t1[3404] := 0.0261197;
   t1[3405] := -0.006971;
   t1[3406] := -0.0028388;
   t1[3407] := 0.002006;
   t1[3408] := 0.0075342;
   t1[3409] := 0.0137687;
   t1[3410] := 0.0207511;
   t1[3411] := 0.0285231;
   t1[3412] := 0.0371264;
   t1[3413] := 0.0465951;
   t1[3414] := 0.0565834;
   t1[3415] := 0.066197;
   t1[3416] := 0.0744987;
   t1[3417] := 0.0805513;
   t1[3418] := 0.0834176;
   t1[3419] := 0.0823831;
   t1[3420] := 0.0848062;
   t1[3421] := 0.0933019;
   t1[3422] := 0.1038192;
   t1[3423] := 0.1163654;
   t1[3424] := 0.129741;
   t1[3425] := 0.1423202;
   t1[3426] := 0.1524764;
   t1[3427] := 0.1585831;
   t1[3428] := 0.1590322;
   t1[3429] := 0.1531259;
   t1[3430] := 0.1414827;
   t1[3431] := 0.1248238;
   t1[3432] := 0.1038702;
   t1[3433] := 0.079343;
   t1[3434] := 0.051917;
   t1[3435] := 0.111939;
   t1[3436] := 0.1034281;
   t1[3437] := 0.0964404;
   t1[3438] := 0.0925468;
   t1[3439] := 0.0919316;
   t1[3440] := 0.0942889;
   t1[3441] := 0.0993123;
   t1[3442] := 0.1066954;
   t1[3443] := 0.1161324;
   t1[3444] := 0.1273434;
   t1[3445] := 0.1400861;
   t1[3446] := 0.1541212;
   t1[3447] := 0.1692092;
   t1[3448] := 0.1851109;
   t1[3449] := 0.2013785;
   t1[3450] := 0.0447403;
   t1[3451] := 0.0547939;
   t1[3452] := 0.0612253;
   t1[3453] := 0.0624766;
   t1[3454] := 0.0588768;
   t1[3455] := 0.0514213;
   t1[3456] := 0.0411066;
   t1[3457] := 0.0289289;
   t1[3458] := 0.0158761;
   t1[3459] := 0.0025055;
   t1[3460] := -0.0112474;
   t1[3461] := -0.0254958;
   t1[3462] := -0.0403527;
   t1[3463] := -0.0559314;
   t1[3464] := -0.0723073;
   t1[3465] := 0.0805147;
   t1[3466] := 0.0761421;
   t1[3467] := 0.0698416;
   t1[3468] := 0.0617641;
   t1[3469] := 0.0522759;
   t1[3470] := 0.0418191;
   t1[3471] := 0.0308362;
   t1[3472] := 0.0197694;
   t1[3473] := 0.0090645;
   t1[3474] := -0.0006555;
   t1[3475] := -0.0085114;
   t1[3476] := -0.0136043;
   t1[3477] := -0.0150351;
   t1[3478] := -0.0119048;
   t1[3479] := -0.0036624;
   t1[3480] := 0.040711;
   t1[3481] := 0.025436;
   t1[3482] := 0.0152156;
   t1[3483] := 0.0117488;
   t1[3484] := 0.0150273;
   t1[3485] := 0.0244397;
   t1[3486] := 0.0393738;
   t1[3487] := 0.0592173;
   t1[3488] := 0.0833447;
   t1[3489] := 0.1104545;
   t1[3490] := 0.1382685;
   t1[3491] := 0.1644324;
   t1[3492] := 0.1865919;
   t1[3493] := 0.2023927;
   t1[3494] := 0.2098137;
   t1[3495] := 0.1020539;
   t1[3496] := 0.110267;
   t1[3497] := 0.1188985;
   t1[3498] := 0.1267664;
   t1[3499] := 0.1333658;
   t1[3500] := 0.1384312;
   t1[3501] := 0.1416971;
   t1[3502] := 0.1428982;
   t1[3503] := 0.1417667;
   t1[3504] := 0.1379156;
   t1[3505] := 0.1307857;
   t1[3506] := 0.1198043;
   t1[3507] := 0.1043986;
   t1[3508] := 0.0839959;
   t1[3509] := 0.0583126;
   t1[3510] := 0.0534281;
   t1[3511] := 0.0553376;
   t1[3512] := 0.0478367;
   t1[3513] := 0.0312592;
   t1[3514] := 0.0076354;
   t1[3515] := -0.0204049;
   t1[3516] := -0.050231;
   t1[3517] := -0.0792125;
   t1[3518] := -0.1047399;
   t1[3519] := -0.1252659;
   t1[3520] := -0.1407779;
   t1[3521] := -0.1513833;
   t1[3522] := -0.1571894;
   t1[3523] := -0.1583035;
   t1[3524] := -0.1548933;
   t1[3525] := 0.1147228;
   t1[3526] := 0.1027995;
   t1[3527] := 0.0950208;
   t1[3528] := 0.0922361;
   t1[3529] := 0.0921171;
   t1[3530] := 0.0912123;
   t1[3531] := 0.0860691;
   t1[3532] := 0.0732349;
   t1[3533] := 0.0493156;
   t1[3534] := 0.0138474;
   t1[3535] := -0.0293984;
   t1[3536] := -0.0763203;
   t1[3537] := -0.1228163;
   t1[3538] := -0.1647848;
   t1[3539] := -0.1985289;
   t1[3540] := 0.2925694;
   t1[3541] := 0.2527561;
   t1[3542] := 0.2060653;
   t1[3543] := 0.1531686;
   t1[3544] := 0.0959583;
   t1[3545] := 0.0367581;
   t1[3546] := -0.0221077;
   t1[3547] := -0.078315;
   t1[3548] := -0.1295486;
   t1[3549] := -0.1739543;
   t1[3550] := -0.2103435;
   t1[3551] := -0.2375795;
   t1[3552] := -0.2545258;
   t1[3553] := -0.2600457;
   t1[3554] := -0.2533901;
   t1[3555] := 0.0990308;
   t1[3556] := 0.0889974;
   t1[3557] := 0.0866131;
   t1[3558] := 0.0937378;
   t1[3559] := 0.107246;
   t1[3560] := 0.1222508;
   t1[3561] := 0.1338631;
   t1[3562] := 0.137194;
   t1[3563] := 0.1274373;
   t1[3564] := 0.1039332;
   t1[3565] := 0.0720146;
   t1[3566] := 0.0374821;
   t1[3567] := 0.0061362;
   t1[3568] := -0.0162224;
   t1[3569] := -0.0247578;
   t1[3570] := 0.0398388;
   t1[3571] := 0.0414079;
   t1[3572] := 0.0459997;
   t1[3573] := 0.0545416;
   t1[3574] := 0.0657353;
   t1[3575] := 0.0774958;
   t1[3576] := 0.087737;
   t1[3577] := 0.094373;
   t1[3578] := 0.0953517;
   t1[3579] := 0.0903113;
   t1[3580] := 0.0813329;
   t1[3581] := 0.0706887;
   t1[3582] := 0.0606504;
   t1[3583] := 0.0534902;
   t1[3584] := 0.0511072;
   t1[3585] := 0.1944849;
   t1[3586] := 0.1775464;
   t1[3587] := 0.155957;
   t1[3588] := 0.1291897;
   t1[3589] := 0.0970577;
   t1[3590] := 0.0594946;
   t1[3591] := 0.0164339;
   t1[3592] := -0.0321907;
   t1[3593] := -0.0864154;
   t1[3594] := -0.1447695;
   t1[3595] := -0.2036044;
   t1[3596] := -0.2591014;
   t1[3597] := -0.3074419;
   t1[3598] := -0.3448073;
   t1[3599] := -0.367875;
   t1[3600] := -0.0492453;
   t1[3601] := -0.0766407;
   t1[3602] := -0.0877784;
   t1[3603] := -0.0788377;
   t1[3604] := -0.0517545;
   t1[3605] := -0.0104991;
   t1[3606] := 0.0409562;
   t1[3607] := 0.0986389;
   t1[3608] := 0.1585754;
   t1[3609] := 0.2167398;
   t1[3610] := 0.2690303;
   t1[3611] := 0.311339;
   t1[3612] := 0.3395582;
   t1[3613] := 0.3495804;
   t1[3614] := 0.3382789;
   t1[3615] := -0.0001066;
   t1[3616] := -0.0023272;
   t1[3617] := 0.0007856;
   t1[3618] := 0.0125822;
   t1[3619] := 0.0319044;
   t1[3620] := 0.0560009;
   t1[3621] := 0.0821188;
   t1[3622] := 0.107505;
   t1[3623] := 0.1294366;
   t1[3624] := 0.1466962;
   t1[3625] := 0.1602426;
   t1[3626] := 0.1712041;
   t1[3627] := 0.1807095;
   t1[3628] := 0.1898872;
   t1[3629] := 0.1995562;
   t1[3630] := 0.1981985;
   t1[3631] := 0.1735667;
   t1[3632] := 0.1448815;
   t1[3633] := 0.1125003;
   t1[3634] := 0.0774915;
   t1[3635] := 0.0411743;
   t1[3636] := 0.0048684;
   t1[3637] := -0.0301067;
   t1[3638] := -0.0624329;
   t1[3639] := -0.0908827;
   t1[3640] := -0.1143581;
   t1[3641] := -0.1317718;
   t1[3642] := -0.1420361;
   t1[3643] := -0.1440635;
   t1[3644] := -0.1371205;
   t1[3645] := 0.3170015;
   t1[3646] := 0.2616679;
   t1[3647] := 0.2037709;
   t1[3648] := 0.1470137;
   t1[3649] := 0.0927804;
   t1[3650] := 0.0416358;
   t1[3651] := -0.0058566;
   t1[3652] := -0.0491329;
   t1[3653] := -0.0876258;
   t1[3654] := -0.1205833;
   t1[3655] := -0.1469865;
   t1[3656] := -0.1657961;
   t1[3657] := -0.1759725;
   t1[3658] := -0.1764761;
   t1[3659] := -0.1666606;
   t1[3660] := -0.1577427;
   t1[3661] := -0.1471254;
   t1[3662] := -0.1316555;
   t1[3663] := -0.1097249;
   t1[3664] := -0.081194;
   t1[3665] := -0.046442;
   t1[3666] := -0.0058484;
   t1[3667] := 0.0402069;
   t1[3668] := 0.0913075;
   t1[3669] := 0.1451974;
   t1[3670] := 0.1969624;
   t1[3671] := 0.2414807;
   t1[3672] := 0.2736304;
   t1[3673] := 0.2882897;
   t1[3674] := 0.2814254;
   t1[3675] := -0.0172095;
   t1[3676] := -0.0105101;
   t1[3677] := -0.0053301;
   t1[3678] := -0.0011242;
   t1[3679] := 0.0029221;
   t1[3680] := 0.0077179;
   t1[3681] := 0.0141728;
   t1[3682] := 0.0231963;
   t1[3683] := 0.0356754;
   t1[3684] := 0.0513815;
   t1[3685] := 0.0684725;
   t1[3686] := 0.0849807;
   t1[3687] := 0.0989384;
   t1[3688] := 0.1083779;
   t1[3689] := 0.1116452;
   t1[3690] := -0.0682686;
   t1[3691] := -0.037591;
   t1[3692] := -0.0066014;
   t1[3693] := 0.0244674;
   t1[3694] := 0.0554993;
   t1[3695] := 0.0864191;
   t1[3696] := 0.117152;
   t1[3697] := 0.147623;
   t1[3698] := 0.1777425;
   t1[3699] := 0.2066816;
   t1[3700] := 0.2325436;
   t1[3701] := 0.2533481;
   t1[3702] := 0.2671148;
   t1[3703] := 0.2718637;
   t1[3704] := 0.2660305;
   t1[3705] := -0.0456219;
   t1[3706] := -0.0433441;
   t1[3707] := -0.0415274;
   t1[3708] := -0.0391814;
   t1[3709] := -0.0357671;
   t1[3710] := -0.030905;
   t1[3711] := -0.0242157;
   t1[3712] := -0.0153201;
   t1[3713] := -0.0038508;
   t1[3714] := 0.0099569;
   t1[3715] := 0.0249969;
   t1[3716] := 0.0400953;
   t1[3717] := 0.054078;
   t1[3718] := 0.0657712;
   t1[3719] := 0.0741331;
   t1[3720] := -0.0242813;
   t1[3721] := -0.0065466;
   t1[3722] := 0.0137707;
   t1[3723] := 0.0359591;
   t1[3724] := 0.0589625;
   t1[3725] := 0.0816028;
   t1[3726] := 0.1027017;
   t1[3727] := 0.121081;
   t1[3728] := 0.1355767;
   t1[3729] := 0.1457374;
   t1[3730] := 0.1521414;
   t1[3731] := 0.1554477;
   t1[3732] := 0.1563148;
   t1[3733] := 0.1554017;
   t1[3734] := 0.1532693;
   t1[3735] := -0.0133028;
   t1[3736] := 0.0137409;
   t1[3737] := 0.0400114;
   t1[3738] := 0.0653678;
   t1[3739] := 0.0894808;
   t1[3740] := 0.1119549;
   t1[3741] := 0.1323943;
   t1[3742] := 0.1504034;
   t1[3743] := 0.1655869;
   t1[3744] := 0.1775824;
   t1[3745] := 0.1860747;
   t1[3746] := 0.1907519;
   t1[3747] := 0.1913026;
   t1[3748] := 0.187415;
   t1[3749] := 0.1788992;
   t1[3750] := 0.0403417;
   t1[3751] := 0.0734304;
   t1[3752] := 0.0977516;
   t1[3753] := 0.1105897;
   t1[3754] := 0.1136943;
   t1[3755] := 0.1103932;
   t1[3756] := 0.1040157;
   t1[3757] := 0.0978914;
   t1[3758] := 0.095308;
   t1[3759] := 0.0974646;
   t1[3760] := 0.1025422;
   t1[3761] := 0.1084861;
   t1[3762] := 0.1132415;
   t1[3763] := 0.1147538;
   t1[3764] := 0.1112914;
   t1[3765] := -0.0214621;
   t1[3766] := -0.0048379;
   t1[3767] := 0.0087356;
   t1[3768] := 0.0179048;
   t1[3769] := 0.0237591;
   t1[3770] := 0.0282516;
   t1[3771] := 0.0333359;
   t1[3772] := 0.0409659;
   t1[3773] := 0.0530614;
   t1[3774] := 0.0698392;
   t1[3775] := 0.0890549;
   t1[3776] := 0.108272;
   t1[3777] := 0.1250539;
   t1[3778] := 0.1369642;
   t1[3779] := 0.1419307;
   t1[3780] := 0.2303855;
   t1[3781] := 0.2239766;
   t1[3782] := 0.2076288;
   t1[3783] := 0.1799457;
   t1[3784] := 0.1435049;
   t1[3785] := 0.1022885;
   t1[3786] := 0.0602801;
   t1[3787] := 0.0214633;
   t1[3788] := -0.0102317;
   t1[3789] := -0.0335598;
   t1[3790] := -0.0511556;
   t1[3791] := -0.0659567;
   t1[3792] := -0.0809006;
   t1[3793] := -0.098925;
   t1[3794] := -0.122269;
   t1[3795] := 0.3787612;
   t1[3796] := 0.321413;
   t1[3797] := 0.2632984;
   t1[3798] := 0.2089968;
   t1[3799] := 0.1576416;
   t1[3800] := 0.1064425;
   t1[3801] := 0.0526067;
   t1[3802] := -0.0066586;
   t1[3803] := -0.0740744;
   t1[3804] := -0.1487714;
   t1[3805] := -0.2246916;
   t1[3806] := -0.2953722;
   t1[3807] := -0.3543501;
   t1[3808] := -0.3951623;
